KUKA KRL program: ps_b_lta_geo_c03.src, ps_b_lta_geo_c03.dat

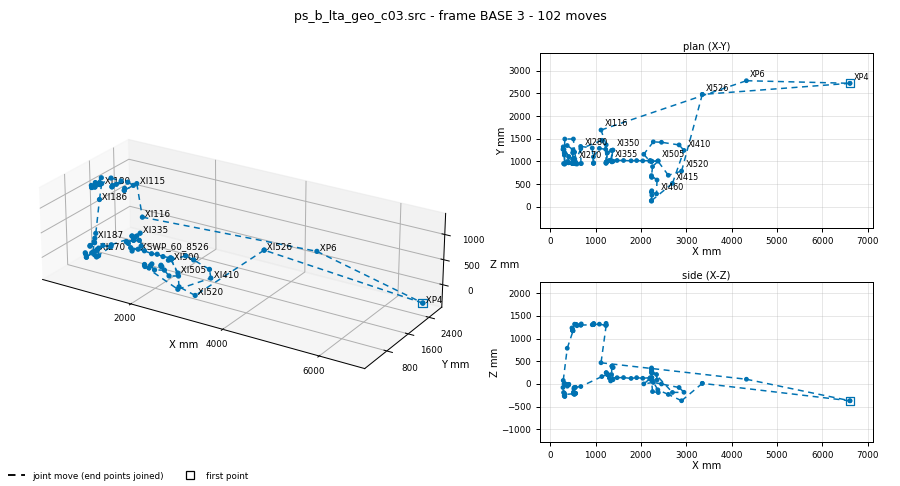
[picture p0: tool path of ps_b_lta_geo_c03.src in frame BASE 3, 102 of 102 moves have a stored position in this frame; points joined in program order, loops and branches not executed]
--- ps_b_lta_geo_c03.src ---
&ACCESS RVO1
&COMMENT Solda Atego LTB
&PARAM DISKPATH = KRC:\R1\Program\OLP
DEF ps_b_lta_geo_c03( )
;FOLD INI
;FOLD SPOTTECH INI
USERSPOT(#INIT)
;ENDFOLD (SPOTTECH INI)
;FOLD GRIPPERTECH INI
USER_GRP(0,DUMMY,DUMMY,GDEFAULT)
;ENDFOLD (GRIPPERTECH INI)
  ;FOLD USER INI
    ;Make your modifications here

  ;ENDFOLD (USER INI)
;ENDFOLD (INI)

; Caracterizacao dos meios de producao
; Changes: Solda Geometria - ATEGO LTB
; Versao Atual:05/01/2016
; Ferramenta: Gun C3
; Name: P13.050-R2
; optimised

chk_w4_wechs_ok( )      ; CHECK GUN C3

;FOLD PTP P4 CONT Vel=100 % PDAT5 Tool[4]:Gun C3 Base[3]:Atego/Axor;%{PE}%R 8.2.20,%MKUKATPBASIS,%CMOVE,%VPTP,%P 1:PTP, 2:P4, 3:C_DIS, 5:100, 7:PDAT5
$BWDSTART=FALSE
PDAT_ACT=PPDAT5
FDAT_ACT=FP4
BAS(#PTP_PARAMS,100)
PTP XP4 C_DIS
;ENDFOLD

if MaxStandMenge (3) then
 MaxStandmengeErreicht (3)
endif

IF (NOT(GHOST())) THEN
if FraesAnf (3) then
 e_fraes4 ()
endif
ENDIF

;FOLD PTP l526 CONT Vel=100 % P_OLP71 Tool[4]:Gun C3 Base[3]:Atego/Axor;%{PE}%R 8.2.20,%MKUKATPBASIS,%CMOVE,%VPTP,%P 1:PTP, 2:l526, 3:C_DIS, 5:100, 7:P_OLP71
$BWDSTART=FALSE
PDAT_ACT=PP_OLP71
FDAT_ACT=Fl526
BAS(#PTP_PARAMS,100)
PTP Xl526 C_DIS
;ENDFOLD

; AGUARDA LIBERACAO PARA SOLDAR GEOMETRIA
;FOLD OUT 3338 'R2 solda geometria Ok' State=FALSE ;%{PE}%R 8.2.20,%MKUKATPBASIS,%COUT,%VOUTX,%P 2:3338, 3:R2 solda geometria Ok, 5:FALSE, 6:
$OUT[3338]=FALSE
;ENDFOLD
;FOLD OUT 3348 'Fora area GEOBOX' State=FALSE ;%{PE}%R 8.2.20,%MKUKATPBASIS,%COUT,%VOUTX,%P 2:3348, 3:Fora area GEOBOX, 5:FALSE, 6:
$OUT[3348]=FALSE
;ENDFOLD
;FOLD OUT 3376 'Lib. p/ soldar Geo Axor/Atego' State=TRUE ;%{PE}%R 8.2.20,%MKUKATPBASIS,%COUT,%VOUTX,%P 2:3376, 3:Lib. p/ soldar Geo Axor/Atego, 5:TRUE, 6:
$OUT[3376]=TRUE
;ENDFOLD
;FOLD WAIT FOR ( IN 3376 'Lib. p/ soldar Geo Axor/Atego' );%{PE}%R 8.2.20,%MKUKATPBASIS,%CEXT_WAIT_FOR,%VEXT_WAIT_FOR,%P 2:, 4:, 5:$IN, 6:3376, 7:Lib. p/ soldar Geo Axor/Atego, 9:
WAIT FOR  ( $IN[3376] )
;ENDFOLD
;FOLD OUT 3376 'Lib. p/ soldar Geo Axor/Atego' State=FALSE ;%{PE}%R 8.2.20,%MKUKATPBASIS,%COUT,%VOUTX,%P 2:3376, 3:Lib. p/ soldar Geo Axor/Atego, 5:FALSE, 6:
$OUT[3376]=FALSE
;ENDFOLD

; LIGA INTERTRAVAMENTO 1 C/ R1
;FOLD Collision.Monitoring_1_On ;%{PE}%MKUKATPUSER
COLLSTOP( 1, 1 ) ;Interrupt-Controlled
;ENDFOLD

; LIGA INTERTRAVAMENTO 4 C/ R4
;FOLD Collision.Monitoring_4_On ;%{PE}%MKUKATPUSER
COLLSTOP( 4, 1 ) ;Interrupt-Controlled
;ENDFOLD

; LIGA INTERTRAVAMENTO 12 C/ R1
;FOLD Collision.Monitoring_AREA_6_On ;%{PE}%MKUKATPUSER
COLLSTOP( 12, 1 ) ;not Interrupt-Controlled
;ENDFOLD

;FOLD PTP l527 CONT Vel=100 % xlarge Tool[4]:Gun C3 Base[3]:Atego/Axor;%{PE}%R 8.2.20,%MKUKATPBASIS,%CMOVE,%VPTP,%P 1:PTP, 2:l527, 3:C_DIS, 5:100, 7:xlarge
$BWDSTART=FALSE
PDAT_ACT=Pxlarge
FDAT_ACT=Fl527
BAS(#PTP_PARAMS,100)
PTP Xl527 C_DIS
;ENDFOLD
;FOLD PTP l520 CONT Vel=100 % xlarge Tool[4]:Gun C3 Base[3]:Atego/Axor;%{PE}%R 8.2.20,%MKUKATPBASIS,%CMOVE,%VPTP,%P 1:PTP, 2:l520, 3:C_DIS, 5:100, 7:xlarge
$BWDSTART=FALSE
PDAT_ACT=Pxlarge
FDAT_ACT=Fl520
BAS(#PTP_PARAMS,100)
PTP Xl520 C_DIS
;ENDFOLD
;FOLD PTP l515 CONT Vel=100 % medium Tool[4]:Gun C3 Base[3]:Atego/Axor;%{PE}%R 8.2.20,%MKUKATPBASIS,%CMOVE,%VPTP,%P 1:PTP, 2:l515, 3:C_DIS, 5:100, 7:medium
$BWDSTART=FALSE
PDAT_ACT=Pmedium
FDAT_ACT=Fl515
BAS(#PTP_PARAMS,100)
PTP Xl515 C_DIS
;ENDFOLD
;FOLD PTP l505 CONT Vel=100 % small Tool[4]:Gun C3 Base[3]:Atego/Axor;%{PE}%R 8.2.20,%MKUKATPBASIS,%CMOVE,%VPTP,%P 1:PTP, 2:l505, 3:C_DIS, 5:100, 7:small
$BWDSTART=FALSE
PDAT_ACT=Psmall
FDAT_ACT=Fl505
BAS(#PTP_PARAMS,100)
PTP Xl505 C_DIS
;ENDFOLD
;FOLD PTP l500 CONT Vel=100 % fin Tool[4]:Gun C3 Base[3]:Atego/Axor;%{PE}%R 8.2.20,%MKUKATPBASIS,%CMOVE,%VPTP,%P 1:PTP, 2:l500, 3:C_DIS, 5:100, 7:fin
$BWDSTART=FALSE
PDAT_ACT=Pfin
FDAT_ACT=Fl500
BAS(#PTP_PARAMS,100)
PTP Xl500 C_DIS
;ENDFOLD

;FOLD ; SWP_60_9492;%{PE}%R 8.2.20,%MKUKATPBASIS,%CCOMMENT,%VNORMAL,%P 2:SWP_60_9492
;ENDFOLD
;FOLD PTP SWP_60_9492 vmax SPOT Gun=3 RETR OPN PgNo1=199 ACTIVE=1 Tool[4]:Gun C3 Base[3]:Atego/Axor;%{PE}%R 8.2.2,%MKUKATPSPOT,%CSPOT,%VPTP,%P 1:PTP, 2:SWP_60_9492, 3:, 5:100, 7:vmax, 10:3, 12:#FIRST, 14:#OPN, 16:199, 18:1, 20:0, 22:0, 24:1, 25:NORMAL
$BWDSTART=FALSE
PDAT_ACT=Pvmax
FDAT_ACT=FSWP_60_9492
BAS(#PTP_PARAMS,Pvmax.VEL)
S_ACT.GUN=3
S_ACT.PAIR=SDEFAULT.PAIR
S_ACT.RETR=#OPN
S_ACT.CLO_TM=1
S_ACT.PGNO1=199
S_ACT.PGNO2=SDEFAULT.PGNO2
S_ACT.PRESS1=SDEFAULT.PRESS1
S_ACT.PRESS2=SDEFAULT.PRESS2
S_READY=FALSE
PTP XSWP_60_9492
USERSPOT(#SPOT, S_ACT)
WAIT FOR S_READY
;ENDFOLD

;FOLD PTP l495 CONT Vel=100 % fin Tool[4]:Gun C3 Base[3]:Atego/Axor;%{PE}%R 8.2.20,%MKUKATPBASIS,%CMOVE,%VPTP,%P 1:PTP, 2:l495, 3:C_DIS, 5:100, 7:fin
$BWDSTART=FALSE
PDAT_ACT=Pfin
FDAT_ACT=Fl495
BAS(#PTP_PARAMS,100)
PTP Xl495 C_DIS
;ENDFOLD
;FOLD PTP l490 CONT Vel=100 % small Tool[4]:Gun C3 Base[3]:Atego/Axor;%{PE}%R 8.2.20,%MKUKATPBASIS,%CMOVE,%VPTP,%P 1:PTP, 2:l490, 3:C_DIS, 5:100, 7:small
$BWDSTART=FALSE
PDAT_ACT=Psmall
FDAT_ACT=Fl490
BAS(#PTP_PARAMS,100)
PTP Xl490 C_DIS
;ENDFOLD
;FOLD PTP l480 CONT Vel=100 % small Tool[4]:Gun C3 Base[3]:Atego/Axor;%{PE}%R 8.2.20,%MKUKATPBASIS,%CMOVE,%VPTP,%P 1:PTP, 2:l480, 3:C_DIS, 5:100, 7:small
$BWDSTART=FALSE
PDAT_ACT=Psmall
FDAT_ACT=Fl480
BAS(#PTP_PARAMS,100)
PTP Xl480 C_DIS
;ENDFOLD
;FOLD PTP l475 CONT Vel=100 % fin Tool[4]:Gun C3 Base[3]:Atego/Axor;%{PE}%R 8.2.20,%MKUKATPBASIS,%CMOVE,%VPTP,%P 1:PTP, 2:l475, 3:C_DIS, 5:100, 7:fin
$BWDSTART=FALSE
PDAT_ACT=Pfin
FDAT_ACT=Fl475
BAS(#PTP_PARAMS,100)
PTP Xl475 C_DIS
;ENDFOLD

;FOLD ; SWP_60_9476;%{PE}%R 8.2.20,%MKUKATPBASIS,%CCOMMENT,%VNORMAL,%P 2:SWP_60_9476
;ENDFOLD
;FOLD PTP SWP_60_9476 vmax SPOT Gun=3 RETR CLS PgNo1=199 ACTIVE=1 Tool[4]:Gun C3 Base[3]:Atego/Axor;%{PE}%R 8.2.2,%MKUKATPSPOT,%CSPOT,%VPTP,%P 1:PTP, 2:SWP_60_9476, 3:, 5:100, 7:vmax, 10:3, 12:#FIRST, 14:#CLO, 16:199, 18:1, 20:0, 22:0, 24:1, 25:NORMAL
$BWDSTART=FALSE
PDAT_ACT=Pvmax
FDAT_ACT=FSWP_60_9476
BAS(#PTP_PARAMS,Pvmax.VEL)
S_ACT.GUN=3
S_ACT.PAIR=SDEFAULT.PAIR
S_ACT.RETR=#CLO
S_ACT.CLO_TM=1
S_ACT.PGNO1=199
S_ACT.PGNO2=SDEFAULT.PGNO2
S_ACT.PRESS1=SDEFAULT.PRESS1
S_ACT.PRESS2=SDEFAULT.PRESS2
S_READY=FALSE
PTP XSWP_60_9476
USERSPOT(#SPOT, S_ACT)
WAIT FOR S_READY
;ENDFOLD

;FOLD PTP l470 CONT Vel=100 % small Tool[4]:Gun C3 Base[3]:Atego/Axor;%{PE}%R 8.2.20,%MKUKATPBASIS,%CMOVE,%VPTP,%P 1:PTP, 2:l470, 3:C_DIS, 5:100, 7:small
$BWDSTART=FALSE
PDAT_ACT=Psmall
FDAT_ACT=Fl470
BAS(#PTP_PARAMS,100)
PTP Xl470 C_DIS
;ENDFOLD
;FOLD PTP l465 CONT Vel=100 % medium Tool[4]:Gun C3 Base[3]:Atego/Axor;%{PE}%R 8.2.20,%MKUKATPBASIS,%CMOVE,%VPTP,%P 1:PTP, 2:l465, 3:C_DIS, 5:100, 7:medium
$BWDSTART=FALSE
PDAT_ACT=Pmedium
FDAT_ACT=Fl465
BAS(#PTP_PARAMS,100)
PTP Xl465 C_DIS
;ENDFOLD
;FOLD PTP l460 CONT Vel=100 % medium Tool[4]:Gun C3 Base[3]:Atego/Axor;%{PE}%R 8.2.20,%MKUKATPBASIS,%CMOVE,%VPTP,%P 1:PTP, 2:l460, 3:C_DIS, 5:100, 7:medium
$BWDSTART=FALSE
PDAT_ACT=Pmedium
FDAT_ACT=Fl460
BAS(#PTP_PARAMS,100)
PTP Xl460 C_DIS
;ENDFOLD
;FOLD PTP l450 CONT Vel=100 % fin Tool[4]:Gun C3 Base[3]:Atego/Axor;%{PE}%R 8.2.20,%MKUKATPBASIS,%CMOVE,%VPTP,%P 1:PTP, 2:l450, 3:C_DIS, 5:100, 7:fin
$BWDSTART=FALSE
PDAT_ACT=Pfin
FDAT_ACT=Fl450
BAS(#PTP_PARAMS,100)
PTP Xl450 C_DIS
;ENDFOLD

;FOLD ; SWP_60_9472;%{PE}%R 8.2.20,%MKUKATPBASIS,%CCOMMENT,%VNORMAL,%P 2:SWP_60_9472
;ENDFOLD
;FOLD PTP SWP_60_9472 vmax SPOT Gun=3 RETR CLS PgNo1=199 ACTIVE=1 Tool[4]:Gun C3 Base[3]:Atego/Axor;%{PE}%R 8.2.2,%MKUKATPSPOT,%CSPOT,%VPTP,%P 1:PTP, 2:SWP_60_9472, 3:, 5:100, 7:vmax, 10:3, 12:#FIRST, 14:#CLO, 16:199, 18:1, 20:0, 22:0, 24:1, 25:NORMAL
$BWDSTART=FALSE
PDAT_ACT=Pvmax
FDAT_ACT=FSWP_60_9472
BAS(#PTP_PARAMS,Pvmax.VEL)
S_ACT.GUN=3
S_ACT.PAIR=SDEFAULT.PAIR
S_ACT.RETR=#CLO
S_ACT.CLO_TM=1
S_ACT.PGNO1=199
S_ACT.PGNO2=SDEFAULT.PGNO2
S_ACT.PRESS1=SDEFAULT.PRESS1
S_ACT.PRESS2=SDEFAULT.PRESS2
S_READY=FALSE
PTP XSWP_60_9472
USERSPOT(#SPOT, S_ACT)
WAIT FOR S_READY
;ENDFOLD


;FOLD PTP l107 CONT Vel=100 % small Tool[4]:Gun C3 Base[3]:Atego/Axor;%{PE}%R 8.2.20,%MKUKATPBASIS,%CMOVE,%VPTP,%P 1:PTP, 2:l107, 3:C_DIS, 5:100, 7:small
$BWDSTART=FALSE
PDAT_ACT=Psmall
FDAT_ACT=Fl107
BAS(#PTP_PARAMS,100)
PTP Xl107 C_DIS
;ENDFOLD
;FOLD PTP l106 CONT Vel=100 % fin Tool[4]:Gun C3 Base[3]:Atego/Axor;%{PE}%R 8.2.20,%MKUKATPBASIS,%CMOVE,%VPTP,%P 1:PTP, 2:l106, 3:C_DIS, 5:100, 7:fin
$BWDSTART=FALSE
PDAT_ACT=Pfin
FDAT_ACT=Fl106
BAS(#PTP_PARAMS,100)
PTP Xl106 C_DIS
;ENDFOLD


;FOLD ; SWP_60_9462;%{PE}%R 8.2.20,%MKUKATPBASIS,%CCOMMENT,%VNORMAL,%P 2:SWP_60_9462
;ENDFOLD
;FOLD PTP SWP_60_9462 vmax SPOT Gun=3 RETR CLS PgNo1=199 ACTIVE=1 Tool[4]:Gun C3 Base[3]:Atego/Axor;%{PE}%R 8.2.2,%MKUKATPSPOT,%CSPOT,%VPTP,%P 1:PTP, 2:SWP_60_9462, 3:, 5:100, 7:vmax, 10:3, 12:#FIRST, 14:#CLO, 16:199, 18:1, 20:0, 22:0, 24:1, 25:NORMAL
$BWDSTART=FALSE
PDAT_ACT=Pvmax
FDAT_ACT=FSWP_60_9462
BAS(#PTP_PARAMS,Pvmax.VEL)
S_ACT.GUN=3
S_ACT.PAIR=SDEFAULT.PAIR
S_ACT.RETR=#CLO
S_ACT.CLO_TM=1
S_ACT.PGNO1=199
S_ACT.PGNO2=SDEFAULT.PGNO2
S_ACT.PRESS1=SDEFAULT.PRESS1
S_ACT.PRESS2=SDEFAULT.PRESS2
S_READY=FALSE
PTP XSWP_60_9462
USERSPOT(#SPOT, S_ACT)
WAIT FOR S_READY
;ENDFOLD

;FOLD PTP l420 CONT Vel=100 % P_OLP48 Tool[4]:Gun C3 Base[3]:Atego/Axor;%{PE}%R 8.2.20,%MKUKATPBASIS,%CMOVE,%VPTP,%P 1:PTP, 2:l420, 3:C_DIS, 5:100, 7:P_OLP48
$BWDSTART=FALSE
PDAT_ACT=PP_OLP48
FDAT_ACT=Fl420
BAS(#PTP_PARAMS,100)
PTP Xl420 C_DIS
;ENDFOLD
;FOLD PTP l415 CONT Vel=100 % xlarge Tool[4]:Gun C3 Base[3]:Atego/Axor;%{PE}%R 8.2.20,%MKUKATPBASIS,%CMOVE,%VPTP,%P 1:PTP, 2:l415, 3:C_DIS, 5:100, 7:xlarge
$BWDSTART=FALSE
PDAT_ACT=Pxlarge
FDAT_ACT=Fl415
BAS(#PTP_PARAMS,100)
PTP Xl415 C_DIS
;ENDFOLD
;FOLD PTP l410 CONT Vel=100 % xlarge Tool[4]:Gun C3 Base[3]:Atego/Axor;%{PE}%R 8.2.20,%MKUKATPBASIS,%CMOVE,%VPTP,%P 1:PTP, 2:l410, 3:C_DIS, 5:100, 7:xlarge
$BWDSTART=FALSE
PDAT_ACT=Pxlarge
FDAT_ACT=Fl410
BAS(#PTP_PARAMS,100)
PTP Xl410 C_DIS
;ENDFOLD
;FOLD PTP l405 CONT Vel=100 % xlarge Tool[4]:Gun C3 Base[3]:Atego/Axor;%{PE}%R 8.2.20,%MKUKATPBASIS,%CMOVE,%VPTP,%P 1:PTP, 2:l405, 3:C_DIS, 5:100, 7:xlarge
$BWDSTART=FALSE
PDAT_ACT=Pxlarge
FDAT_ACT=Fl405
BAS(#PTP_PARAMS,100)
PTP Xl405 C_DIS
;ENDFOLD
;FOLD PTP l400 CONT Vel=100 % medium Tool[4]:Gun C3 Base[3]:Atego/Axor;%{PE}%R 8.2.20,%MKUKATPBASIS,%CMOVE,%VPTP,%P 1:PTP, 2:l400, 3:C_DIS, 5:100, 7:medium
$BWDSTART=FALSE
PDAT_ACT=Pmedium
FDAT_ACT=Fl400
BAS(#PTP_PARAMS,100)
PTP Xl400 C_DIS
;ENDFOLD
;FOLD PTP l395 CONT Vel=100 % xlarge Tool[4]:Gun C3 Base[3]:Atego/Axor;%{PE}%R 8.2.20,%MKUKATPBASIS,%CMOVE,%VPTP,%P 1:PTP, 2:l395, 3:C_DIS, 5:100, 7:xlarge
$BWDSTART=FALSE
PDAT_ACT=Pxlarge
FDAT_ACT=Fl395
BAS(#PTP_PARAMS,100)
PTP Xl395 C_DIS
;ENDFOLD
;FOLD PTP l390 CONT Vel=100 % medium Tool[4]:Gun C3 Base[3]:Atego/Axor;%{PE}%R 8.2.20,%MKUKATPBASIS,%CMOVE,%VPTP,%P 1:PTP, 2:l390, 3:C_DIS, 5:100, 7:medium
$BWDSTART=FALSE
PDAT_ACT=Pmedium
FDAT_ACT=Fl390
BAS(#PTP_PARAMS,100)
PTP Xl390 C_DIS
;ENDFOLD
;FOLD PTP l385 CONT Vel=100 % fin Tool[4]:Gun C3 Base[3]:Atego/Axor;%{PE}%R 8.2.20,%MKUKATPBASIS,%CMOVE,%VPTP,%P 1:PTP, 2:l385, 3:C_DIS, 5:100, 7:fin
$BWDSTART=FALSE
PDAT_ACT=Pfin
FDAT_ACT=Fl385
BAS(#PTP_PARAMS,100)
PTP Xl385 C_DIS
;ENDFOLD

;FOLD ; SWP_60_8494;%{PE}%R 8.2.20,%MKUKATPBASIS,%CCOMMENT,%VNORMAL,%P 2:SWP_60_8494
;ENDFOLD
;FOLD PTP SWP_60_8494 vmax SPOT Gun=3 RETR CLS PgNo1=211 ACTIVE=1 Tool[4]:Gun C3 Base[3]:Atego/Axor;%{PE}%R 8.2.2,%MKUKATPSPOT,%CSPOT,%VPTP,%P 1:PTP, 2:SWP_60_8494, 3:, 5:100, 7:vmax, 10:3, 12:#FIRST, 14:#CLO, 16:211, 18:1, 20:0, 22:0, 24:1, 25:NORMAL
$BWDSTART=FALSE
PDAT_ACT=Pvmax
FDAT_ACT=FSWP_60_8494
BAS(#PTP_PARAMS,Pvmax.VEL)
S_ACT.GUN=3
S_ACT.PAIR=SDEFAULT.PAIR
S_ACT.RETR=#CLO
S_ACT.CLO_TM=1
S_ACT.PGNO1=211
S_ACT.PGNO2=SDEFAULT.PGNO2
S_ACT.PRESS1=SDEFAULT.PRESS1
S_ACT.PRESS2=SDEFAULT.PRESS2
S_READY=FALSE
PTP XSWP_60_8494
USERSPOT(#SPOT, S_ACT)
WAIT FOR S_READY
;ENDFOLD

; DESLIGA INTERTRAVAMENTO 12 C/ R1
;FOLD Collision.Monitoring_AREA_6_Off . ;%{PE}%MKUKATPUSER
COLLSTOP( 12, 2+0 )
;ENDFOLD

;FOLD PTP P5 CONT Vel=100 % large Tool[4]:Gun C3 Base[3]:Atego/Axor;%{PE}%R 8.2.20,%MKUKATPBASIS,%CMOVE,%VPTP,%P 1:PTP, 2:P5, 3:C_DIS, 5:100, 7:large
$BWDSTART=FALSE
PDAT_ACT=Plarge
FDAT_ACT=FP5
BAS(#PTP_PARAMS,100)
PTP XP5 C_DIS
;ENDFOLD

;FOLD ; SWP_60_8506;%{PE}%R 8.2.20,%MKUKATPBASIS,%CCOMMENT,%VNORMAL,%P 2:SWP_60_8506
;ENDFOLD
;FOLD PTP SWP_60_8506 vmax SPOT Gun=3 RETR CLS PgNo1=203 ACTIVE=1 Tool[4]:Gun C3 Base[3]:Atego/Axor;%{PE}%R 8.2.2,%MKUKATPSPOT,%CSPOT,%VPTP,%P 1:PTP, 2:SWP_60_8506, 3:, 5:100, 7:vmax, 10:3, 12:#FIRST, 14:#CLO, 16:203, 18:1, 20:0, 22:0, 24:1, 25:NORMAL
$BWDSTART=FALSE
PDAT_ACT=Pvmax
FDAT_ACT=FSWP_60_8506
BAS(#PTP_PARAMS,Pvmax.VEL)
S_ACT.GUN=3
S_ACT.PAIR=SDEFAULT.PAIR
S_ACT.RETR=#CLO
S_ACT.CLO_TM=1
S_ACT.PGNO1=203
S_ACT.PGNO2=SDEFAULT.PGNO2
S_ACT.PRESS1=SDEFAULT.PRESS1
S_ACT.PRESS2=SDEFAULT.PRESS2
S_READY=FALSE
PTP XSWP_60_8506
USERSPOT(#SPOT, S_ACT)
WAIT FOR S_READY
;ENDFOLD

;FOLD PTP l380 CONT Vel=100 % large Tool[4]:Gun C3 Base[3]:Atego/Axor;%{PE}%R 8.2.20,%MKUKATPBASIS,%CMOVE,%VPTP,%P 1:PTP, 2:l380, 3:C_DIS, 5:100, 7:large
$BWDSTART=FALSE
PDAT_ACT=Plarge
FDAT_ACT=Fl380
BAS(#PTP_PARAMS,100)
PTP Xl380 C_DIS
;ENDFOLD

;FOLD ; SWP_60_8518;%{PE}%R 8.2.20,%MKUKATPBASIS,%CCOMMENT,%VNORMAL,%P 2:SWP_60_8518
;ENDFOLD
;FOLD PTP SWP_60_8518 vmax SPOT Gun=3 RETR CLS PgNo1=212 ACTIVE=1 Tool[4]:Gun C3 Base[3]:Atego/Axor;%{PE}%R 8.2.2,%MKUKATPSPOT,%CSPOT,%VPTP,%P 1:PTP, 2:SWP_60_8518, 3:, 5:100, 7:vmax, 10:3, 12:#FIRST, 14:#CLO, 16:212, 18:1, 20:0, 22:0, 24:1, 25:NORMAL
$BWDSTART=FALSE
PDAT_ACT=Pvmax
FDAT_ACT=FSWP_60_8518
BAS(#PTP_PARAMS,Pvmax.VEL)
S_ACT.GUN=3
S_ACT.PAIR=SDEFAULT.PAIR
S_ACT.RETR=#CLO
S_ACT.CLO_TM=1
S_ACT.PGNO1=212
S_ACT.PGNO2=SDEFAULT.PGNO2
S_ACT.PRESS1=SDEFAULT.PRESS1
S_ACT.PRESS2=SDEFAULT.PRESS2
S_READY=FALSE
PTP XSWP_60_8518
USERSPOT(#SPOT, S_ACT)
WAIT FOR S_READY
;ENDFOLD

;FOLD ; SWP_60_8526;%{PE}%R 8.2.20,%MKUKATPBASIS,%CCOMMENT,%VNORMAL,%P 2:SWP_60_8526
;ENDFOLD
;FOLD PTP SWP_60_8526 vmax SPOT Gun=3 RETR CLS PgNo1=206 ACTIVE=1 Tool[4]:Gun C3 Base[3]:Atego/Axor;%{PE}%R 8.2.2,%MKUKATPSPOT,%CSPOT,%VPTP,%P 1:PTP, 2:SWP_60_8526, 3:, 5:100, 7:vmax, 10:3, 12:#FIRST, 14:#CLO, 16:206, 18:1, 20:0, 22:0, 24:1, 25:NORMAL
$BWDSTART=FALSE
PDAT_ACT=Pvmax
FDAT_ACT=FSWP_60_8526
BAS(#PTP_PARAMS,Pvmax.VEL)
S_ACT.GUN=3
S_ACT.PAIR=SDEFAULT.PAIR
S_ACT.RETR=#CLO
S_ACT.CLO_TM=1
S_ACT.PGNO1=206
S_ACT.PGNO2=SDEFAULT.PGNO2
S_ACT.PRESS1=SDEFAULT.PRESS1
S_ACT.PRESS2=SDEFAULT.PRESS2
S_READY=FALSE
PTP XSWP_60_8526
USERSPOT(#SPOT, S_ACT)
WAIT FOR S_READY
;ENDFOLD

;FOLD ; SWP_60_8534;%{PE}%R 8.2.20,%MKUKATPBASIS,%CCOMMENT,%VNORMAL,%P 2:SWP_60_8534
;ENDFOLD
;FOLD PTP SWP_60_8534 vmax SPOT Gun=3 RETR CLS PgNo1=206 ACTIVE=1 Tool[4]:Gun C3 Base[3]:Atego/Axor;%{PE}%R 8.2.2,%MKUKATPSPOT,%CSPOT,%VPTP,%P 1:PTP, 2:SWP_60_8534, 3:, 5:100, 7:vmax, 10:3, 12:#FIRST, 14:#CLO, 16:206, 18:1, 20:0, 22:0, 24:1, 25:NORMAL
$BWDSTART=FALSE
PDAT_ACT=Pvmax
FDAT_ACT=FSWP_60_8534
BAS(#PTP_PARAMS,Pvmax.VEL)
S_ACT.GUN=3
S_ACT.PAIR=SDEFAULT.PAIR
S_ACT.RETR=#CLO
S_ACT.CLO_TM=1
S_ACT.PGNO1=206
S_ACT.PGNO2=SDEFAULT.PGNO2
S_ACT.PRESS1=SDEFAULT.PRESS1
S_ACT.PRESS2=SDEFAULT.PRESS2
S_READY=FALSE
PTP XSWP_60_8534
USERSPOT(#SPOT, S_ACT)
WAIT FOR S_READY
;ENDFOLD

;FOLD PTP l355 CONT Vel=100 % small Tool[4]:Gun C3 Base[3]:Atego/Axor;%{PE}%R 8.2.20,%MKUKATPBASIS,%CMOVE,%VPTP,%P 1:PTP, 2:l355, 3:C_DIS, 5:100, 7:small
$BWDSTART=FALSE
PDAT_ACT=Psmall
FDAT_ACT=Fl355
BAS(#PTP_PARAMS,100)
PTP Xl355 C_DIS
;ENDFOLD
;FOLD PTP l350 CONT Vel=100 % large Tool[4]:Gun C3 Base[3]:Atego/Axor;%{PE}%R 8.2.20,%MKUKATPBASIS,%CMOVE,%VPTP,%P 1:PTP, 2:l350, 3:C_DIS, 5:100, 7:large
$BWDSTART=FALSE
PDAT_ACT=Plarge
FDAT_ACT=Fl350
BAS(#PTP_PARAMS,100)
PTP Xl350 C_DIS
;ENDFOLD
;FOLD PTP l335 CONT Vel=100 % medium Tool[4]:Gun C3 Base[3]:Atego/Axor;%{PE}%R 8.2.20,%MKUKATPBASIS,%CMOVE,%VPTP,%P 1:PTP, 2:l335, 3:C_DIS, 5:100, 7:medium
$BWDSTART=FALSE
PDAT_ACT=Pmedium
FDAT_ACT=Fl335
BAS(#PTP_PARAMS,100)
PTP Xl335 C_DIS
;ENDFOLD
;FOLD PTP l330 CONT Vel=100 % fin Tool[4]:Gun C3 Base[3]:Atego/Axor;%{PE}%R 8.2.20,%MKUKATPBASIS,%CMOVE,%VPTP,%P 1:PTP, 2:l330, 3:C_DIS, 5:100, 7:fin
$BWDSTART=FALSE
PDAT_ACT=Pfin
FDAT_ACT=Fl330
BAS(#PTP_PARAMS,100)
PTP Xl330 C_DIS
;ENDFOLD

;FOLD ; SWP_60_8554;%{PE}%R 8.2.20,%MKUKATPBASIS,%CCOMMENT,%VNORMAL,%P 2:SWP_60_8554
;ENDFOLD
;FOLD PTP SWP_60_8554 vmax SPOT Gun=3 RETR CLS PgNo1=197 ACTIVE=1 Tool[4]:Gun C3 Base[3]:Atego/Axor;%{PE}%R 8.2.2,%MKUKATPSPOT,%CSPOT,%VPTP,%P 1:PTP, 2:SWP_60_8554, 3:, 5:100, 7:vmax, 10:3, 12:#FIRST, 14:#CLO, 16:197, 18:1, 20:0, 22:0, 24:1, 25:NORMAL
$BWDSTART=FALSE
PDAT_ACT=Pvmax
FDAT_ACT=FSWP_60_8554
BAS(#PTP_PARAMS,Pvmax.VEL)
S_ACT.GUN=3
S_ACT.PAIR=SDEFAULT.PAIR
S_ACT.RETR=#CLO
S_ACT.CLO_TM=1
S_ACT.PGNO1=197
S_ACT.PGNO2=SDEFAULT.PGNO2
S_ACT.PRESS1=SDEFAULT.PRESS1
S_ACT.PRESS2=SDEFAULT.PRESS2
S_READY=FALSE
PTP XSWP_60_8554
USERSPOT(#SPOT, S_ACT)
WAIT FOR S_READY
;ENDFOLD

;FOLD PTP l325 CONT Vel=100 % fin Tool[4]:Gun C3 Base[3]:Atego/Axor;%{PE}%R 8.2.20,%MKUKATPBASIS,%CMOVE,%VPTP,%P 1:PTP, 2:l325, 3:C_DIS, 5:100, 7:fin
$BWDSTART=FALSE
PDAT_ACT=Pfin
FDAT_ACT=Fl325
BAS(#PTP_PARAMS,100)
PTP Xl325 C_DIS
;ENDFOLD
;FOLD PTP l320 CONT Vel=100 % small Tool[4]:Gun C3 Base[3]:Atego/Axor;%{PE}%R 8.2.20,%MKUKATPBASIS,%CMOVE,%VPTP,%P 1:PTP, 2:l320, 3:C_DIS, 5:100, 7:small
$BWDSTART=FALSE
PDAT_ACT=Psmall
FDAT_ACT=Fl320
BAS(#PTP_PARAMS,100)
PTP Xl320 C_DIS
;ENDFOLD
;FOLD PTP l310 CONT Vel=100 % small Tool[4]:Gun C3 Base[3]:Atego/Axor;%{PE}%R 8.2.20,%MKUKATPBASIS,%CMOVE,%VPTP,%P 1:PTP, 2:l310, 3:C_DIS, 5:100, 7:small
$BWDSTART=FALSE
PDAT_ACT=Psmall
FDAT_ACT=Fl310
BAS(#PTP_PARAMS,100)
PTP Xl310 C_DIS
;ENDFOLD
;FOLD PTP l300 CONT Vel=100 % fin Tool[4]:Gun C3 Base[3]:Atego/Axor;%{PE}%R 8.2.20,%MKUKATPBASIS,%CMOVE,%VPTP,%P 1:PTP, 2:l300, 3:C_DIS, 5:100, 7:fin
$BWDSTART=FALSE
PDAT_ACT=Pfin
FDAT_ACT=Fl300
BAS(#PTP_PARAMS,100)
PTP Xl300 C_DIS
;ENDFOLD

;FOLD ; SWP_60_8542;%{PE}%R 8.2.20,%MKUKATPBASIS,%CCOMMENT,%VNORMAL,%P 2:SWP_60_8542
;ENDFOLD
;FOLD PTP SWP_60_8542 vmax SPOT Gun=3 RETR CLS PgNo1=215 ACTIVE=1 Tool[4]:Gun C3 Base[3]:Atego/Axor;%{PE}%R 8.2.2,%MKUKATPSPOT,%CSPOT,%VPTP,%P 1:PTP, 2:SWP_60_8542, 3:, 5:100, 7:vmax, 10:3, 12:#FIRST, 14:#CLO, 16:215, 18:1, 20:0, 22:0, 24:1, 25:NORMAL
$BWDSTART=FALSE
PDAT_ACT=Pvmax
FDAT_ACT=FSWP_60_8542
BAS(#PTP_PARAMS,Pvmax.VEL)
S_ACT.GUN=3
S_ACT.PAIR=SDEFAULT.PAIR
S_ACT.RETR=#CLO
S_ACT.CLO_TM=1
S_ACT.PGNO1=215
S_ACT.PGNO2=SDEFAULT.PGNO2
S_ACT.PRESS1=SDEFAULT.PRESS1
S_ACT.PRESS2=SDEFAULT.PRESS2
S_READY=FALSE
PTP XSWP_60_8542
USERSPOT(#SPOT, S_ACT)
WAIT FOR S_READY
;ENDFOLD

;FOLD PTP l295 CONT Vel=100 % fin Tool[4]:Gun C3 Base[3]:Atego/Axor;%{PE}%R 8.2.20,%MKUKATPBASIS,%CMOVE,%VPTP,%P 1:PTP, 2:l295, 3:C_DIS, 5:100, 7:fin
$BWDSTART=FALSE
PDAT_ACT=Pfin
FDAT_ACT=Fl295
BAS(#PTP_PARAMS,100)
PTP Xl295 C_DIS
;ENDFOLD
;FOLD PTP l290 CONT Vel=100 % small Tool[4]:Gun C3 Base[3]:Atego/Axor;%{PE}%R 8.2.20,%MKUKATPBASIS,%CMOVE,%VPTP,%P 1:PTP, 2:l290, 3:C_DIS, 5:100, 7:small
$BWDSTART=FALSE
PDAT_ACT=Psmall
FDAT_ACT=Fl290
BAS(#PTP_PARAMS,100)
PTP Xl290 C_DIS
;ENDFOLD
;FOLD PTP l285 CONT Vel=100 % large Tool[4]:Gun C3 Base[3]:Atego/Axor;%{PE}%R 8.2.20,%MKUKATPBASIS,%CMOVE,%VPTP,%P 1:PTP, 2:l285, 3:C_DIS, 5:100, 7:large
$BWDSTART=FALSE
PDAT_ACT=Plarge
FDAT_ACT=Fl285
BAS(#PTP_PARAMS,100)
PTP Xl285 C_DIS
;ENDFOLD
;FOLD PTP l280 CONT Vel=100 % medium Tool[4]:Gun C3 Base[3]:Atego/Axor;%{PE}%R 8.2.20,%MKUKATPBASIS,%CMOVE,%VPTP,%P 1:PTP, 2:l280, 3:C_DIS, 5:100, 7:medium
$BWDSTART=FALSE
PDAT_ACT=Pmedium
FDAT_ACT=Fl280
BAS(#PTP_PARAMS,100)
PTP Xl280 C_DIS
;ENDFOLD
;FOLD PTP l270 CONT Vel=100 % fin Tool[4]:Gun C3 Base[3]:Atego/Axor;%{PE}%R 8.2.20,%MKUKATPBASIS,%CMOVE,%VPTP,%P 1:PTP, 2:l270, 3:C_DIS, 5:100, 7:fin
$BWDSTART=FALSE
PDAT_ACT=Pfin
FDAT_ACT=Fl270
BAS(#PTP_PARAMS,100)
PTP Xl270 C_DIS
;ENDFOLD

;FOLD ; SWP_60_8068;%{PE}%R 8.2.20,%MKUKATPBASIS,%CCOMMENT,%VNORMAL,%P 2:SWP_60_8068
;ENDFOLD
;FOLD PTP SWP_60_8068 fin SPOT Gun=3 RETR CLS PgNo1=207 ACTIVE=1 Tool[4]:Gun C3 Base[3]:Atego/Axor;%{PE}%R 8.2.2,%MKUKATPSPOT,%CSPOT,%VPTP,%P 1:PTP, 2:SWP_60_8068, 3:, 5:100, 7:fin, 10:3, 12:#FIRST, 14:#CLO, 16:207, 18:1, 20:0, 22:0, 24:1, 25:NORMAL
$BWDSTART=FALSE
PDAT_ACT=Pfin
FDAT_ACT=FSWP_60_8068
BAS(#PTP_PARAMS,Pfin.VEL)
S_ACT.GUN=3
S_ACT.PAIR=SDEFAULT.PAIR
S_ACT.RETR=#CLO
S_ACT.CLO_TM=1
S_ACT.PGNO1=207
S_ACT.PGNO2=SDEFAULT.PGNO2
S_ACT.PRESS1=SDEFAULT.PRESS1
S_ACT.PRESS2=SDEFAULT.PRESS2
S_READY=FALSE
PTP XSWP_60_8068
USERSPOT(#SPOT, S_ACT)
WAIT FOR S_READY
;ENDFOLD

;FOLD PTP l265 CONT Vel=100 % fin Tool[4]:Gun C3 Base[3]:Atego/Axor;%{PE}%R 8.2.20,%MKUKATPBASIS,%CMOVE,%VPTP,%P 1:PTP, 2:l265, 3:C_DIS, 5:100, 7:fin
$BWDSTART=FALSE
PDAT_ACT=Pfin
FDAT_ACT=Fl265
BAS(#PTP_PARAMS,100)
PTP Xl265 C_DIS
;ENDFOLD
;FOLD PTP l255 CONT Vel=100 % small Tool[4]:Gun C3 Base[3]:Atego/Axor;%{PE}%R 8.2.20,%MKUKATPBASIS,%CMOVE,%VPTP,%P 1:PTP, 2:l255, 3:C_DIS, 5:100, 7:small
$BWDSTART=FALSE
PDAT_ACT=Psmall
FDAT_ACT=Fl255
BAS(#PTP_PARAMS,100)
PTP Xl255 C_DIS
;ENDFOLD
;FOLD PTP l250 CONT Vel=100 % small Tool[4]:Gun C3 Base[3]:Atego/Axor;%{PE}%R 8.2.20,%MKUKATPBASIS,%CMOVE,%VPTP,%P 1:PTP, 2:l250, 3:C_DIS, 5:100, 7:small
$BWDSTART=FALSE
PDAT_ACT=Psmall
FDAT_ACT=Fl250
BAS(#PTP_PARAMS,100)
PTP Xl250 C_DIS
;ENDFOLD
;FOLD PTP l240 CONT Vel=100 % fin Tool[4]:Gun C3 Base[3]:Atego/Axor;%{PE}%R 8.2.20,%MKUKATPBASIS,%CMOVE,%VPTP,%P 1:PTP, 2:l240, 3:C_DIS, 5:100, 7:fin
$BWDSTART=FALSE
PDAT_ACT=Pfin
FDAT_ACT=Fl240
BAS(#PTP_PARAMS,100)
PTP Xl240 C_DIS
;ENDFOLD

;FOLD ; SWP_60_8060;%{PE}%R 8.2.20,%MKUKATPBASIS,%CCOMMENT,%VNORMAL,%P 2:SWP_60_8060
;ENDFOLD
;FOLD PTP SWP_60_8060 vmax SPOT Gun=3 RETR OPN PgNo1=210 ACTIVE=1 Tool[4]:Gun C3 Base[3]:Atego/Axor;%{PE}%R 8.2.2,%MKUKATPSPOT,%CSPOT,%VPTP,%P 1:PTP, 2:SWP_60_8060, 3:, 5:100, 7:vmax, 10:3, 12:#FIRST, 14:#OPN, 16:210, 18:1, 20:0, 22:0, 24:1, 25:NORMAL
$BWDSTART=FALSE
PDAT_ACT=Pvmax
FDAT_ACT=FSWP_60_8060
BAS(#PTP_PARAMS,Pvmax.VEL)
S_ACT.GUN=3
S_ACT.PAIR=SDEFAULT.PAIR
S_ACT.RETR=#OPN
S_ACT.CLO_TM=1
S_ACT.PGNO1=210
S_ACT.PGNO2=SDEFAULT.PGNO2
S_ACT.PRESS1=SDEFAULT.PRESS1
S_ACT.PRESS2=SDEFAULT.PRESS2
S_READY=FALSE
PTP XSWP_60_8060
USERSPOT(#SPOT, S_ACT)
WAIT FOR S_READY
;ENDFOLD

;FOLD PTP l230 CONT Vel=100 % fin Tool[4]:Gun C3 Base[3]:Atego/Axor;%{PE}%R 8.2.20,%MKUKATPBASIS,%CMOVE,%VPTP,%P 1:PTP, 2:l230, 3:C_DIS, 5:100, 7:fin
$BWDSTART=FALSE
PDAT_ACT=Pfin
FDAT_ACT=Fl230
BAS(#PTP_PARAMS,100)
PTP Xl230 C_DIS
;ENDFOLD
;FOLD PTP l225 CONT Vel=100 % medium Tool[4]:Gun C3 Base[3]:Atego/Axor;%{PE}%R 8.2.20,%MKUKATPBASIS,%CMOVE,%VPTP,%P 1:PTP, 2:l225, 3:C_DIS, 5:100, 7:medium
$BWDSTART=FALSE
PDAT_ACT=Pmedium
FDAT_ACT=Fl225
BAS(#PTP_PARAMS,100)
PTP Xl225 C_DIS
;ENDFOLD
;FOLD PTP l220 CONT Vel=100 % medium Tool[4]:Gun C3 Base[3]:Atego/Axor;%{PE}%R 8.2.20,%MKUKATPBASIS,%CMOVE,%VPTP,%P 1:PTP, 2:l220, 3:C_DIS, 5:100, 7:medium
$BWDSTART=FALSE
PDAT_ACT=Pmedium
FDAT_ACT=Fl220
BAS(#PTP_PARAMS,100)
PTP Xl220 C_DIS
;ENDFOLD
;FOLD PTP l215 CONT Vel=100 % small Tool[4]:Gun C3 Base[3]:Atego/Axor;%{PE}%R 8.2.20,%MKUKATPBASIS,%CMOVE,%VPTP,%P 1:PTP, 2:l215, 3:C_DIS, 5:100, 7:small
$BWDSTART=FALSE
PDAT_ACT=Psmall
FDAT_ACT=Fl215
BAS(#PTP_PARAMS,100)
PTP Xl215 C_DIS
;ENDFOLD
;FOLD PTP l210 CONT Vel=100 % small Tool[4]:Gun C3 Base[3]:Atego/Axor;%{PE}%R 8.2.20,%MKUKATPBASIS,%CMOVE,%VPTP,%P 1:PTP, 2:l210, 3:C_DIS, 5:100, 7:small
$BWDSTART=FALSE
PDAT_ACT=Psmall
FDAT_ACT=Fl210
BAS(#PTP_PARAMS,100)
PTP Xl210 C_DIS
;ENDFOLD
;FOLD PTP l205 CONT Vel=100 % fin Tool[4]:Gun C3 Base[3]:Atego/Axor;%{PE}%R 8.2.20,%MKUKATPBASIS,%CMOVE,%VPTP,%P 1:PTP, 2:l205, 3:C_DIS, 5:100, 7:fin
$BWDSTART=FALSE
PDAT_ACT=Pfin
FDAT_ACT=Fl205
BAS(#PTP_PARAMS,100)
PTP Xl205 C_DIS
;ENDFOLD

;FOLD ; SWP_60_8046;%{PE}%R 8.2.20,%MKUKATPBASIS,%CCOMMENT,%VNORMAL,%P 2:SWP_60_8046
;ENDFOLD
;FOLD PTP SWP_60_8046 fin SPOT Gun=3 RETR OPN PgNo1=202 ACTIVE=1 Tool[4]:Gun C3 Base[3]:Atego/Axor;%{PE}%R 8.2.2,%MKUKATPSPOT,%CSPOT,%VPTP,%P 1:PTP, 2:SWP_60_8046, 3:, 5:100, 7:fin, 10:3, 12:#FIRST, 14:#OPN, 16:202, 18:1, 20:0, 22:0, 24:1, 25:NORMAL
$BWDSTART=FALSE
PDAT_ACT=Pfin
FDAT_ACT=FSWP_60_8046
BAS(#PTP_PARAMS,Pfin.VEL)
S_ACT.GUN=3
S_ACT.PAIR=SDEFAULT.PAIR
S_ACT.RETR=#OPN
S_ACT.CLO_TM=1
S_ACT.PGNO1=202
S_ACT.PGNO2=SDEFAULT.PGNO2
S_ACT.PRESS1=SDEFAULT.PRESS1
S_ACT.PRESS2=SDEFAULT.PRESS2
S_READY=FALSE
PTP XSWP_60_8046
USERSPOT(#SPOT, S_ACT)
WAIT FOR S_READY
;ENDFOLD

;FOLD PTP l200 CONT Vel=100 % fin Tool[4]:Gun C3 Base[3]:Atego/Axor;%{PE}%R 8.2.20,%MKUKATPBASIS,%CMOVE,%VPTP,%P 1:PTP, 2:l200, 3:C_DIS, 5:100, 7:fin
$BWDSTART=FALSE
PDAT_ACT=Pfin
FDAT_ACT=Fl200
BAS(#PTP_PARAMS,100)
PTP Xl200 C_DIS
;ENDFOLD
;FOLD PTP l195 CONT Vel=100 % medium Tool[4]:Gun C3 Base[3]:Atego/Axor;%{PE}%R 8.2.20,%MKUKATPBASIS,%CMOVE,%VPTP,%P 1:PTP, 2:l195, 3:C_DIS, 5:100, 7:medium
$BWDSTART=FALSE
PDAT_ACT=Pmedium
FDAT_ACT=Fl195
BAS(#PTP_PARAMS,100)
PTP Xl195 C_DIS
;ENDFOLD
;FOLD PTP l185 CONT Vel=100 % medium Tool[4]:Gun C3 Base[3]:Atego/Axor;%{PE}%R 8.2.20,%MKUKATPBASIS,%CMOVE,%VPTP,%P 1:PTP, 2:l185, 3:C_DIS, 5:100, 7:medium
$BWDSTART=FALSE
PDAT_ACT=Pmedium
FDAT_ACT=Fl185
BAS(#PTP_PARAMS,100)
PTP Xl185 C_DIS
;ENDFOLD
;FOLD PTP l187 CONT Vel=100 % medium Tool[4]:Gun C3 Base[3]:Atego/Axor;%{PE}%R 8.2.20,%MKUKATPBASIS,%CMOVE,%VPTP,%P 1:PTP, 2:l187, 3:C_DIS, 5:100, 7:medium
$BWDSTART=FALSE
PDAT_ACT=Pmedium
FDAT_ACT=Fl187
BAS(#PTP_PARAMS,100)
PTP Xl187 C_DIS
;ENDFOLD
;FOLD PTP l036 CONT Vel=100 % medium Tool[4]:Gun C3 Base[3]:Atego/Axor;%{PE}%R 8.2.20,%MKUKATPBASIS,%CMOVE,%VPTP,%P 1:PTP, 2:l036, 3:C_DIS, 5:100, 7:medium
$BWDSTART=FALSE
PDAT_ACT=Pmedium
FDAT_ACT=Fl036
BAS(#PTP_PARAMS,100)
PTP Xl036 C_DIS
;ENDFOLD
;FOLD PTP l031 CONT Vel=100 % fin Tool[4]:Gun C3 Base[3]:Atego/Axor;%{PE}%R 8.2.20,%MKUKATPBASIS,%CMOVE,%VPTP,%P 1:PTP, 2:l031, 3:C_DIS, 5:100, 7:fin
$BWDSTART=FALSE
PDAT_ACT=Pfin
FDAT_ACT=Fl031
BAS(#PTP_PARAMS,100)
PTP Xl031 C_DIS
;ENDFOLD

;FOLD ; SWP_60_9078;%{PE}%R 8.2.20,%MKUKATPBASIS,%CCOMMENT,%VNORMAL,%P 2:SWP_60_9078
;ENDFOLD
;FOLD PTP SWP_60_9078 vmax SPOT Gun=3 RETR CLS PgNo1=213 ACTIVE=1 Tool[4]:Gun C3 Base[3]:Atego/Axor;%{PE}%R 8.2.2,%MKUKATPSPOT,%CSPOT,%VPTP,%P 1:PTP, 2:SWP_60_9078, 3:, 5:100, 7:vmax, 10:3, 12:#FIRST, 14:#CLO, 16:213, 18:1, 20:0, 22:0, 24:1, 25:NORMAL
$BWDSTART=FALSE
PDAT_ACT=Pvmax
FDAT_ACT=FSWP_60_9078
BAS(#PTP_PARAMS,Pvmax.VEL)
S_ACT.GUN=3
S_ACT.PAIR=SDEFAULT.PAIR
S_ACT.RETR=#CLO
S_ACT.CLO_TM=1
S_ACT.PGNO1=213
S_ACT.PGNO2=SDEFAULT.PGNO2
S_ACT.PRESS1=SDEFAULT.PRESS1
S_ACT.PRESS2=SDEFAULT.PRESS2
S_READY=FALSE
PTP XSWP_60_9078
USERSPOT(#SPOT, S_ACT)
WAIT FOR S_READY
;ENDFOLD

;FOLD PTP l026 CONT Vel=100 % fin Tool[4]:Gun C3 Base[3]:Atego/Axor;%{PE}%R 8.2.20,%MKUKATPBASIS,%CMOVE,%VPTP,%P 1:PTP, 2:l026, 3:C_DIS, 5:100, 7:fin
$BWDSTART=FALSE
PDAT_ACT=Pfin
FDAT_ACT=Fl026
BAS(#PTP_PARAMS,100)
PTP Xl026 C_DIS
;ENDFOLD
;FOLD PTP l021 CONT Vel=100 % medium Tool[4]:Gun C3 Base[3]:Atego/Axor;%{PE}%R 8.2.20,%MKUKATPBASIS,%CMOVE,%VPTP,%P 1:PTP, 2:l021, 3:C_DIS, 5:100, 7:medium
$BWDSTART=FALSE
PDAT_ACT=Pmedium
FDAT_ACT=Fl021
BAS(#PTP_PARAMS,100)
PTP Xl021 C_DIS
;ENDFOLD
;FOLD PTP l188 CONT Vel=100 % medium Tool[4]:Gun C3 Base[3]:Atego/Axor;%{PE}%R 8.2.20,%MKUKATPBASIS,%CMOVE,%VPTP,%P 1:PTP, 2:l188, 3:C_DIS, 5:100, 7:medium
$BWDSTART=FALSE
PDAT_ACT=Pmedium
FDAT_ACT=Fl188
BAS(#PTP_PARAMS,100)
PTP Xl188 C_DIS
;ENDFOLD
;FOLD PTP l186 CONT Vel=100 % large Tool[4]:Gun C3 Base[3]:Atego/Axor;%{PE}%R 8.2.20,%MKUKATPBASIS,%CMOVE,%VPTP,%P 1:PTP, 2:l186, 3:C_DIS, 5:100, 7:large
$BWDSTART=FALSE
PDAT_ACT=Plarge
FDAT_ACT=Fl186
BAS(#PTP_PARAMS,100)
PTP Xl186 C_DIS
;ENDFOLD
;FOLD PTP l180 CONT Vel=100 % medium Tool[4]:Gun C3 Base[3]:Atego/Axor;%{PE}%R 8.2.20,%MKUKATPBASIS,%CMOVE,%VPTP,%P 1:PTP, 2:l180, 3:C_DIS, 5:100, 7:medium
$BWDSTART=FALSE
PDAT_ACT=Pmedium
FDAT_ACT=Fl180
BAS(#PTP_PARAMS,100)
PTP Xl180 C_DIS
;ENDFOLD
;FOLD PTP l175 CONT Vel=100 % small Tool[4]:Gun C3 Base[3]:Atego/Axor;%{PE}%R 8.2.20,%MKUKATPBASIS,%CMOVE,%VPTP,%P 1:PTP, 2:l175, 3:C_DIS, 5:100, 7:small
$BWDSTART=FALSE
PDAT_ACT=Psmall
FDAT_ACT=Fl175
BAS(#PTP_PARAMS,100)
PTP Xl175 C_DIS
;ENDFOLD
;FOLD PTP l170 CONT Vel=100 % fin Tool[4]:Gun C3 Base[3]:Atego/Axor;%{PE}%R 8.2.20,%MKUKATPBASIS,%CMOVE,%VPTP,%P 1:PTP, 2:l170, 3:C_DIS, 5:100, 7:fin
$BWDSTART=FALSE
PDAT_ACT=Pfin
FDAT_ACT=Fl170
BAS(#PTP_PARAMS,100)
PTP Xl170 C_DIS
;ENDFOLD

;FOLD ; SWP_60_8576;%{PE}%R 8.2.20,%MKUKATPBASIS,%CCOMMENT,%VNORMAL,%P 2:SWP_60_8576
;ENDFOLD
;FOLD PTP SWP_60_8576 vmax SPOT Gun=3 RETR CLS PgNo1=209 ACTIVE=1 Tool[4]:Gun C3 Base[3]:Atego/Axor;%{PE}%R 8.2.2,%MKUKATPSPOT,%CSPOT,%VPTP,%P 1:PTP, 2:SWP_60_8576, 3:, 5:100, 7:vmax, 10:3, 12:#FIRST, 14:#CLO, 16:209, 18:1, 20:0, 22:0, 24:1, 25:NORMAL
$BWDSTART=FALSE
PDAT_ACT=Pvmax
FDAT_ACT=FSWP_60_8576
BAS(#PTP_PARAMS,Pvmax.VEL)
S_ACT.GUN=3
S_ACT.PAIR=SDEFAULT.PAIR
S_ACT.RETR=#CLO
S_ACT.CLO_TM=1
S_ACT.PGNO1=209
S_ACT.PGNO2=SDEFAULT.PGNO2
S_ACT.PRESS1=SDEFAULT.PRESS1
S_ACT.PRESS2=SDEFAULT.PRESS2
S_READY=FALSE
PTP XSWP_60_8576
USERSPOT(#SPOT, S_ACT)
WAIT FOR S_READY
;ENDFOLD

;FOLD PTP l171 CONT Vel=100 % fin Tool[4]:Gun C3 Base[3]:Atego/Axor;%{PE}%R 8.2.20,%MKUKATPBASIS,%CMOVE,%VPTP,%P 1:PTP, 2:l171, 3:C_DIS, 5:100, 7:fin
$BWDSTART=FALSE
PDAT_ACT=Pfin
FDAT_ACT=Fl171
BAS(#PTP_PARAMS,100)
PTP Xl171 C_DIS
;ENDFOLD
;FOLD PTP l160 CONT Vel=100 % medium Tool[4]:Gun C3 Base[3]:Atego/Axor;%{PE}%R 8.2.20,%MKUKATPBASIS,%CMOVE,%VPTP,%P 1:PTP, 2:l160, 3:C_DIS, 5:100, 7:medium
$BWDSTART=FALSE
PDAT_ACT=Pmedium
FDAT_ACT=Fl160
BAS(#PTP_PARAMS,100)
PTP Xl160 C_DIS
;ENDFOLD
;FOLD PTP l155 CONT Vel=100 % mediun Tool[4]:Gun C3 Base[3]:Atego/Axor;%{PE}%R 8.2.20,%MKUKATPBASIS,%CMOVE,%VPTP,%P 1:PTP, 2:l155, 3:C_DIS, 5:100, 7:mediun
$BWDSTART=FALSE
PDAT_ACT=Pmediun
FDAT_ACT=Fl155
BAS(#PTP_PARAMS,100)
PTP Xl155 C_DIS
;ENDFOLD
;FOLD PTP l157 CONT Vel=100 % small Tool[4]:Gun C3 Base[3]:Atego/Axor;%{PE}%R 8.2.20,%MKUKATPBASIS,%CMOVE,%VPTP,%P 1:PTP, 2:l157, 3:C_DIS, 5:100, 7:small
$BWDSTART=FALSE
PDAT_ACT=Psmall
FDAT_ACT=Fl157
BAS(#PTP_PARAMS,100)
PTP Xl157 C_DIS
;ENDFOLD
;FOLD PTP l158 CONT Vel=100 % fin Tool[4]:Gun C3 Base[3]:Atego/Axor;%{PE}%R 8.2.20,%MKUKATPBASIS,%CMOVE,%VPTP,%P 1:PTP, 2:l158, 3:C_DIS, 5:100, 7:fin
$BWDSTART=FALSE
PDAT_ACT=Pfin
FDAT_ACT=Fl158
BAS(#PTP_PARAMS,100)
PTP Xl158 C_DIS
;ENDFOLD

;FOLD ; SWP_60_8584;%{PE}%R 8.2.20,%MKUKATPBASIS,%CCOMMENT,%VNORMAL,%P 2:SWP_60_8584
;ENDFOLD
;FOLD PTP SWP_60_8584 vmax SPOT Gun=3 RETR CLS PgNo1=200 ACTIVE=1 Tool[4]:Gun C3 Base[3]:Atego/Axor;%{PE}%R 8.2.2,%MKUKATPSPOT,%CSPOT,%VPTP,%P 1:PTP, 2:SWP_60_8584, 3:, 5:100, 7:vmax, 10:3, 12:#FIRST, 14:#CLO, 16:200, 18:1, 20:0, 22:0, 24:1, 25:NORMAL
$BWDSTART=FALSE
PDAT_ACT=Pvmax
FDAT_ACT=FSWP_60_8584
BAS(#PTP_PARAMS,Pvmax.VEL)
S_ACT.GUN=3
S_ACT.PAIR=SDEFAULT.PAIR
S_ACT.RETR=#CLO
S_ACT.CLO_TM=1
S_ACT.PGNO1=200
S_ACT.PGNO2=SDEFAULT.PGNO2
S_ACT.PRESS1=SDEFAULT.PRESS1
S_ACT.PRESS2=SDEFAULT.PRESS2
S_READY=FALSE
PTP XSWP_60_8584
USERSPOT(#SPOT, S_ACT)
WAIT FOR S_READY
;ENDFOLD

;FOLD ; SWP_60_8788;%{PE}%R 8.2.20,%MKUKATPBASIS,%CCOMMENT,%VNORMAL,%P 2:SWP_60_8788
;ENDFOLD
;FOLD PTP SWP_60_8788 vmax SPOT Gun=3 RETR CLS PgNo1=200 ACTIVE=1 Tool[4]:Gun C3 Base[3]:Atego/Axor;%{PE}%R 8.2.2,%MKUKATPSPOT,%CSPOT,%VPTP,%P 1:PTP, 2:SWP_60_8788, 3:, 5:100, 7:vmax, 10:3, 12:#FIRST, 14:#CLO, 16:200, 18:1, 20:0, 22:0, 24:1, 25:NORMAL
$BWDSTART=FALSE
PDAT_ACT=Pvmax
FDAT_ACT=FSWP_60_8788
BAS(#PTP_PARAMS,Pvmax.VEL)
S_ACT.GUN=3
S_ACT.PAIR=SDEFAULT.PAIR
S_ACT.RETR=#CLO
S_ACT.CLO_TM=1
S_ACT.PGNO1=200
S_ACT.PGNO2=SDEFAULT.PGNO2
S_ACT.PRESS1=SDEFAULT.PRESS1
S_ACT.PRESS2=SDEFAULT.PRESS2
S_READY=FALSE
PTP XSWP_60_8788
USERSPOT(#SPOT, S_ACT)
WAIT FOR S_READY
;ENDFOLD

;FOLD PTP l159 CONT Vel=100 % fin Tool[4]:Gun C3 Base[3]:Atego/Axor;%{PE}%R 8.2.20,%MKUKATPBASIS,%CMOVE,%VPTP,%P 1:PTP, 2:l159, 3:C_DIS, 5:100, 7:fin
$BWDSTART=FALSE
PDAT_ACT=Pfin
FDAT_ACT=Fl159
BAS(#PTP_PARAMS,100)
PTP Xl159 C_DIS
;ENDFOLD
;FOLD PTP l161 CONT Vel=100 % medium Tool[4]:Gun C3 Base[3]:Atego/Axor;%{PE}%R 8.2.20,%MKUKATPBASIS,%CMOVE,%VPTP,%P 1:PTP, 2:l161, 3:C_DIS, 5:100, 7:medium
$BWDSTART=FALSE
PDAT_ACT=Pmedium
FDAT_ACT=Fl161
BAS(#PTP_PARAMS,100)
PTP Xl161 C_DIS
;ENDFOLD
;FOLD PTP l162 CONT Vel=100 % medium Tool[4]:Gun C3 Base[3]:Atego/Axor;%{PE}%R 8.2.20,%MKUKATPBASIS,%CMOVE,%VPTP,%P 1:PTP, 2:l162, 3:C_DIS, 5:100, 7:medium
$BWDSTART=FALSE
PDAT_ACT=Pmedium
FDAT_ACT=Fl162
BAS(#PTP_PARAMS,100)
PTP Xl162 C_DIS
;ENDFOLD
;FOLD PTP l163 CONT Vel=100 % fin Tool[4]:Gun C3 Base[3]:Atego/Axor;%{PE}%R 8.2.20,%MKUKATPBASIS,%CMOVE,%VPTP,%P 1:PTP, 2:l163, 3:C_DIS, 5:100, 7:fin
$BWDSTART=FALSE
PDAT_ACT=Pfin
FDAT_ACT=Fl163
BAS(#PTP_PARAMS,100)
PTP Xl163 C_DIS
;ENDFOLD

;FOLD ; SWP_60_8800;%{PE}%R 8.2.20,%MKUKATPBASIS,%CCOMMENT,%VNORMAL,%P 2:SWP_60_8800
;ENDFOLD
;FOLD PTP SWP_60_8800 vmax SPOT Gun=3 RETR CLS PgNo1=196 ACTIVE=1 Tool[4]:Gun C3 Base[3]:Atego/Axor;%{PE}%R 8.2.2,%MKUKATPSPOT,%CSPOT,%VPTP,%P 1:PTP, 2:SWP_60_8800, 3:, 5:100, 7:vmax, 10:3, 12:#FIRST, 14:#CLO, 16:196, 18:1, 20:0, 22:0, 24:1, 25:NORMAL
$BWDSTART=FALSE
PDAT_ACT=Pvmax
FDAT_ACT=FSWP_60_8800
BAS(#PTP_PARAMS,Pvmax.VEL)
S_ACT.GUN=3
S_ACT.PAIR=SDEFAULT.PAIR
S_ACT.RETR=#CLO
S_ACT.CLO_TM=1
S_ACT.PGNO1=196
S_ACT.PGNO2=SDEFAULT.PGNO2
S_ACT.PRESS1=SDEFAULT.PRESS1
S_ACT.PRESS2=SDEFAULT.PRESS2
S_READY=FALSE
PTP XSWP_60_8800
USERSPOT(#SPOT, S_ACT)
WAIT FOR S_READY
;ENDFOLD

;FOLD PTP l164 CONT Vel=100 % fin Tool[4]:Gun C3 Base[3]:Atego/Axor;%{PE}%R 8.2.20,%MKUKATPBASIS,%CMOVE,%VPTP,%P 1:PTP, 2:l164, 3:C_DIS, 5:100, 7:fin
$BWDSTART=FALSE
PDAT_ACT=Pfin
FDAT_ACT=Fl164
BAS(#PTP_PARAMS,100)
PTP Xl164 C_DIS
;ENDFOLD
;FOLD PTP l166 CONT Vel=100 % small Tool[4]:Gun C3 Base[3]:Atego/Axor;%{PE}%R 8.2.20,%MKUKATPBASIS,%CMOVE,%VPTP,%P 1:PTP, 2:l166, 3:C_DIS, 5:100, 7:small
$BWDSTART=FALSE
PDAT_ACT=Psmall
FDAT_ACT=Fl166
BAS(#PTP_PARAMS,100)
PTP Xl166 C_DIS
;ENDFOLD
;FOLD PTP l150 CONT Vel=100 % small Tool[4]:Gun C3 Base[3]:Atego/Axor;%{PE}%R 8.2.20,%MKUKATPBASIS,%CMOVE,%VPTP,%P 1:PTP, 2:l150, 3:C_DIS, 5:100, 7:small
$BWDSTART=FALSE
PDAT_ACT=Psmall
FDAT_ACT=Fl150
BAS(#PTP_PARAMS,100)
PTP Xl150 C_DIS
;ENDFOLD
;FOLD PTP l145 CONT Vel=100 % small Tool[4]:Gun C3 Base[3]:Atego/Axor;%{PE}%R 8.2.20,%MKUKATPBASIS,%CMOVE,%VPTP,%P 1:PTP, 2:l145, 3:C_DIS, 5:100, 7:small
$BWDSTART=FALSE
PDAT_ACT=Psmall
FDAT_ACT=Fl145
BAS(#PTP_PARAMS,100)
PTP Xl145 C_DIS
;ENDFOLD
;FOLD PTP l135 CONT Vel=100 % fin Tool[4]:Gun C3 Base[3]:Atego/Axor;%{PE}%R 8.2.20,%MKUKATPBASIS,%CMOVE,%VPTP,%P 1:PTP, 2:l135, 3:C_DIS, 5:100, 7:fin
$BWDSTART=FALSE
PDAT_ACT=Pfin
FDAT_ACT=Fl135
BAS(#PTP_PARAMS,100)
PTP Xl135 C_DIS
;ENDFOLD

;FOLD ; SWP_60_8812;%{PE}%R 8.2.20,%MKUKATPBASIS,%CCOMMENT,%VNORMAL,%P 2:SWP_60_8812
;ENDFOLD
;FOLD PTP SWP_60_8812 vmax SPOT Gun=3 RETR OPN PgNo1=207 ACTIVE=1 Tool[4]:Gun C3 Base[3]:Atego/Axor;%{PE}%R 8.2.2,%MKUKATPSPOT,%CSPOT,%VPTP,%P 1:PTP, 2:SWP_60_8812, 3:, 5:100, 7:vmax, 10:3, 12:#FIRST, 14:#OPN, 16:207, 18:1, 20:0, 22:0, 24:1, 25:NORMAL
$BWDSTART=FALSE
PDAT_ACT=Pvmax
FDAT_ACT=FSWP_60_8812
BAS(#PTP_PARAMS,Pvmax.VEL)
S_ACT.GUN=3
S_ACT.PAIR=SDEFAULT.PAIR
S_ACT.RETR=#OPN
S_ACT.CLO_TM=1
S_ACT.PGNO1=207
S_ACT.PGNO2=SDEFAULT.PGNO2
S_ACT.PRESS1=SDEFAULT.PRESS1
S_ACT.PRESS2=SDEFAULT.PRESS2
S_READY=FALSE
PTP XSWP_60_8812
USERSPOT(#SPOT, S_ACT)
WAIT FOR S_READY
;ENDFOLD

;FOLD PTP l130 CONT Vel=100 % fin Tool[4]:Gun C3 Base[3]:Atego/Axor;%{PE}%R 8.2.20,%MKUKATPBASIS,%CMOVE,%VPTP,%P 1:PTP, 2:l130, 3:C_DIS, 5:100, 7:fin
$BWDSTART=FALSE
PDAT_ACT=Pfin
FDAT_ACT=Fl130
BAS(#PTP_PARAMS,100)
PTP Xl130 C_DIS
;ENDFOLD
;FOLD PTP l115 CONT Vel=100 % medium Tool[4]:Gun C3 Base[3]:Atego/Axor;%{PE}%R 8.2.20,%MKUKATPBASIS,%CMOVE,%VPTP,%P 1:PTP, 2:l115, 3:C_DIS, 5:100, 7:medium
$BWDSTART=FALSE
PDAT_ACT=Pmedium
FDAT_ACT=Fl115
BAS(#PTP_PARAMS,100)
PTP Xl115 C_DIS
;ENDFOLD
;FOLD PTP l116 Vel=100 % vmax Tool[4]:Gun C3 Base[3]:Atego/Axor;%{PE}%R 8.2.20,%MKUKATPBASIS,%CMOVE,%VPTP,%P 1:PTP, 2:l116, 3:, 5:100, 7:vmax
$BWDSTART=FALSE
PDAT_ACT=Pvmax
FDAT_ACT=Fl116
BAS(#PTP_PARAMS,100)
PTP Xl116
;ENDFOLD

; FIM DE TRABALHO GEOMETRIA
;FOLD PULSE 3338 'R2 solda geometria Ok' State=TRUE Time=3 sec;%{PE}%R 8.2.20,%MKUKATPBASIS,%COUT,%VPULSE,%P 2:3338, 3:R2 solda geometria Ok, 5:TRUE, 6:, 8:3
PULSE($OUT[3338], TRUE,3)
;ENDFOLD
;FOLD OUT 3348 'Fora area GEOBOX' State=TRUE ;%{PE}%R 8.2.20,%MKUKATPBASIS,%COUT,%VOUTX,%P 2:3348, 3:Fora area GEOBOX, 5:TRUE, 6:
$OUT[3348]=TRUE
;ENDFOLD

; DESLIGA INTERTRAVAMENTO 1 C/ R1
;FOLD Collision.Monitoring_1_Off . ;%{PE}%MKUKATPUSER
COLLSTOP( 1, 2+0 )
;ENDFOLD

; DESLIGA INTERTRAVAMENTO 4 C/ R4
;FOLD Collision.Monitoring_4_Off . ;%{PE}%MKUKATPUSER
COLLSTOP( 4, 2+0 )
;ENDFOLD

; LIGA INTERLOCK 5 C/ R5
;FOLD Collision.Monitoring_5_On ;%{PE}%MKUKATPUSER
COLLSTOP( 5, 1 ) ;not Interrupt-Controlled
;ENDFOLD

;FOLD PTP P6 CONT Vel=100 % xxlarge Tool[4]:Gun C3 Base[3]:Atego/Axor;%{PE}%R 8.2.20,%MKUKATPBASIS,%CMOVE,%VPTP,%P 1:PTP, 2:P6, 3:C_DIS, 5:100, 7:xxlarge
$BWDSTART=FALSE
PDAT_ACT=Pxxlarge
FDAT_ACT=FP6
BAS(#PTP_PARAMS,100)
PTP XP6 C_DIS
;ENDFOLD
;FOLD PTP P3 Vel=100 % vmax Tool[4]:Gun C3 Base[3]:Atego/Axor;%{PE}%R 8.2.20,%MKUKATPBASIS,%CMOVE,%VPTP,%P 1:PTP, 2:P3, 3:, 5:100, 7:vmax
$BWDSTART=FALSE
PDAT_ACT=Pvmax
FDAT_ACT=FP3
BAS(#PTP_PARAMS,100)
PTP XP3
;ENDFOLD

IF (NOT(GHOST())) THEN
if FraesAnf (3) then
 f_fraes4 ()
endif
ENDIF

END

--- ps_b_lta_geo_c03.dat ---
&ACCESS RVO1
&COMMENT Solda Atego LTB
&PARAM DISKPATH = KRC:\R1\Program\OLP
DEFDAT ps_b_lta_geo_c03
;FOLD EXTERNAL DECLARATIONS;%{PE}%MKUKATPBASIS,%CEXT,%VCOMMON,%P
;FOLD GRIPPERTECH EXT
EXT  H50 (INT  :IN,INT  :IN,INT  :IN,GRP_TYP  :IN )
;ENDFOLD (GRIPPERTECH EXT)
;FOLD SPOTTECH EXT
EXT  USERSPOT (S_COMMAND  :IN,SPOT_TYPE  :IN )
;ENDFOLD (SPOTTECH EXT)
;FOLD BASISTECH EXT;%{PE}%MKUKATPBASIS,%CEXT,%VEXT,%P
EXT  BAS (BAS_COMMAND  :IN,REAL  :IN )
DECL INT SUCCESS
;ENDFOLD (BASISTECH EXT)
;FOLD USER EXT;%{E}%MKUKATPUSER,%CEXT,%VEXT,%P
;Make your modifications here

;ENDFOLD (USER EXT)
;ENDFOLD (EXTERNAL DECLARATIONS)



DECL PDAT PP_OLP4={VEL 100.0,ACC 100.0,APO_DIST 20.0,APO_MODE #CDIS}
DECL PDAT PP_OLP7={VEL 100.0,ACC 100.0,APO_DIST 100.0,APO_MODE #CDIS}


; E6POS declarations
; FDAT declarations
; LDAT declarations
; PDAT declarations

; E6POS declarations
DECL E6POS XSWP_60_9078={X 377.429504,Y 998.692078,Z -51.6705818,A -178.750397,B 54.3092003,C 89.6855087,S 2,T 11,E1 -5500.00195,E2 0.0,E3 0.0,E4 0.0,E5 0.0,E6 0.0}
DECL E6POS XSWP_60_8584={X 574.901672,Y 959.645203,Z 1312.65002,A -171.738693,B -53.4007301,C 82.1439133,S 2,T 11,E1 -5500.0,E2 0.0,E3 0.0,E4 0.0,E5 0.0,E6 0.0}
DECL E6POS XSWP_60_8788={X 685.193909,Y 955.620117,Z 1322.33398,A -124.007103,B -84.2773209,C 35.6398811,S 2,T 11,E1 -5500.0,E2 0.0,E3 0.0,E4 0.0,E5 0.0,E6 0.0}
DECL E6POS XSWP_60_8800={X 959.385071,Y 969.231201,Z 1333.18396,A -9.99958229,B -68.941597,C -77.7464828,S 2,T 11,E1 -5500.0,E2 0.0,E3 0.0,E4 0.0,E5 0.0,E6 0.0}
DECL E6POS Xl115={X 1235.03198,Y 1367.06604,Z 1292.71497,A -80.0313873,B -85.9020309,C -9.10745239,S 2,T 10,E1 -5500.0,E2 0.0,E3 0.0,E4 0.0,E5 0.0,E6 0.0}
DECL E6POS Xl130={X 1231.23999,Y 962.339111,Z 1297.51001,A -81.1379089,B -84.6478424,C -7.77770805,S 2,T 11,E1 -5499.99902,E2 0.0,E3 0.0,E4 0.0,E5 0.0,E6 0.0}
DECL E6POS XSWP_60_8812={X 1232.76001,Y 973.570801,Z 1334.12903,A -79.7475128,B -85.9006195,C -9.10391426,S 2,T 11,E1 -5499.99902,E2 0.0,E3 0.0,E4 0.0,E5 0.0,E6 0.0}
DECL E6POS Xl135={X 1231.23999,Y 962.339111,Z 1297.51001,A -81.1379089,B -84.6478424,C -7.77770805,S 2,T 11,E1 -5499.99902,E2 0.0,E3 0.0,E4 0.0,E5 0.0,E6 0.0}
DECL E6POS Xl145={X 1225.06006,Y 1267.27502,Z 1289.97595,A -82.990799,B -85.3915329,C -5.86582804,S 2,T 10,E1 -5500.0,E2 0.0,E3 0.0,E4 0.0,E5 0.0,E6 0.0}
DECL E6POS Xl150={X 1084.92798,Y 1289.59802,Z 1316.64697,A -110.132202,B -85.2466202,C 21.2871304,S 2,T 10,E1 -5500.0,E2 0.0,E3 0.0,E4 0.0,E5 0.0,E6 0.0}
DECL E6POS Xl155={X 495.042297,Y 1192.729,Z 1176.08704,A -166.6194,B -62.0061798,C 77.3858871,S 2,T 10,E1 -5500.0,E2 0.0,E3 0.0,E4 0.0,E5 0.0,E6 0.0}
DECL E6POS Xl160={X 495.625793,Y 1048.98596,Z 1173.58606,A -166.463699,B -59.9506111,C 75.8885117,S 2,T 11,E1 -5500.0,E2 0.0,E3 0.0,E4 0.0,E5 0.0,E6 0.0}
DECL E6POS XSWP_60_8576={X 479.7323,Y 961.704895,Z 1232.96802,A -168.522095,B -65.2164001,C 79.4213181,S 2,T 11,E1 -5500.0,E2 0.0,E3 0.0,E4 0.0,E5 0.0,E6 0.0}
DECL E6POS Xl170={X 493.426605,Y 954.01123,Z 1196.677,A -165.408203,B -64.9694595,C 76.488472,S 2,T 11,E1 -5500.0,E2 0.0,E3 0.0,E4 0.0,E5 0.0,E6 0.0}
DECL E6POS Xl175={X 498.414612,Y 1048.99402,Z 1175.27905,A -167.799103,B -56.2781601,C 76.6106262,S 2,T 11,E1 -5500.0,E2 0.0,E3 0.0,E4 0.0,E5 0.0,E6 0.0}
DECL E6POS Xl180={X 504.707489,Y 1257.96997,Z 1171.14404,A -175.011902,B -65.2939529,C 85.5748062,S 2,T 10,E1 -5500.0,E2 0.0,E3 0.0,E4 0.0,E5 0.0,E6 0.0}
DECL E6POS Xl185={X 281.523285,Y 1267.26001,Z -80.7737808,A -171.102203,B -55.8212395,C 78.1676636,S 2,T 10,E1 -5500.00195,E2 0.0,E3 0.0,E4 0.0,E5 0.0,E6 0.0}
DECL E6POS Xl195={X 309.236694,Y 1189.24902,Z -261.055695,A -161.565903,B -64.5644531,C 71.0960388,S 2,T 10,E1 -5500.00586,E2 0.0,E3 0.0,E4 0.0,E5 0.0,E6 0.0}
DECL E6POS Xl200={X 320.765808,Y 952.112915,Z -276.100006,A -170.774399,B -65.5663605,C 82.4341507,S 2,T 11,E1 -5500.00586,E2 0.0,E3 0.0,E4 0.0,E5 0.0,E6 0.0}
DECL E6POS XSWP_60_8046={X 295.258392,Y 953.246582,Z -191.709198,A -178.112198,B -65.694397,C 89.5197296,S 2,T 11,E1 -5500.00586,E2 0.0,E3 0.0,E4 0.0,E5 0.0,E6 0.0}
DECL E6POS Xl205={X 313.821808,Y 939.276306,Z -206.506302,A -176.364502,B -65.6938019,C 88.284462,S 2,T 11,E1 -5500.00586,E2 0.0,E3 0.0,E4 0.0,E5 0.0,E6 0.0}
DECL E6POS Xl210={X 320.765808,Y 952.112915,Z -276.100006,A -170.774399,B -65.5663528,C 82.4341507,S 2,T 11,E1 -5500.00586,E2 0.0,E3 0.0,E4 0.0,E5 0.0,E6 0.0}
DECL E6POS Xl215={X 311.768311,Y 1138.82202,Z -260.171997,A -172.248505,B -65.4501114,C 83.7742386,S 2,T 10,E1 -5500.00586,E2 0.0,E3 0.0,E4 0.0,E5 0.0,E6 0.0}
DECL E6POS Xl220={X 321.698212,Y 1495.271,Z -235.324005,A 177.775497,B -76.9053802,C 89.1578827,S 2,T 10,E1 -5500.0,E2 0.0,E3 0.0,E4 0.0,E5 0.0,E6 0.0}
DECL E6POS Xl225={X 511.616211,Y 1495.66797,Z -217.2724,A -176.421494,B -85.6921997,C 87.4376068,S 2,T 10,E1 -5500.0,E2 0.0,E3 0.0,E4 0.0,E5 0.0,E6 0.0}
DECL E6POS Xl230={X 561.25293,Y 949.928406,Z -209.439102,A -162.895203,B -85.5735092,C 75.3529587,S 2,T 11,E1 -5499.99805,E2 0.0,E3 0.0,E4 0.0,E5 0.0,E6 0.0}
DECL E6POS XSWP_60_8060={X 512.477783,Y 955.514282,Z -183.049194,A -176.456406,B -85.6937866,C 87.4698563,S 2,T 11,E1 -5499.99805,E2 0.0,E3 0.0,E4 0.0,E5 0.0,E6 0.0}
DECL E6POS Xl240={X 561.25293,Y 949.928406,Z -209.439102,A -162.895203,B -85.5735092,C 75.3529587,S 2,T 11,E1 -5499.99805,E2 0.0,E3 0.0,E4 0.0,E5 0.0,E6 0.0}
DECL E6POS Xl250={X 534.108521,Y 1051.99402,Z -234.229004,A -178.033707,B -27.6022606,C 88.6840973,S 2,T 11,E1 -5500.0,E2 0.0,E3 0.0,E4 0.0,E5 0.0,E6 0.0}
DECL E6POS Xl255={X 526.619873,Y 1071.71301,Z -83.3147964,A -178.809601,B 34.4082718,C 89.7623367,S 2,T 10,E1 -5500.0,E2 0.0,E3 0.0,E4 0.0,E5 0.0,E6 0.0}
DECL E6POS Xl265={X 552.832581,Y 992.614319,Z -76.7540436,A -177.865707,B 43.6499786,C 90.5385971,S 2,T 11,E1 -5500.00488,E2 0.0,E3 0.0,E4 0.0,E5 0.0,E6 0.0}
DECL E6POS XSWP_60_8068={X 522.917725,Y 999.467896,Z -110.008202,A -178.878799,B 43.6501999,C 89.7160492,S 2,T 11,E1 -5500.00488,E2 0.0,E3 0.0,E4 0.0,E5 0.0,E6 0.0}
DECL E6POS Xl270={X 552.832581,Y 992.614319,Z -76.7540436,A -177.865707,B 43.6499786,C 90.5385971,S 2,T 11,E1 -5500.00488,E2 0.0,E3 0.0,E4 0.0,E5 0.0,E6 0.0}
DECL E6POS Xl280={X 675.09613,Y 1281.73804,Z -58.8733101,A 178.420898,B 65.5474091,C 89.3197327,S 2,T 10,E1 -5500.0,E2 0.0,E3 0.0,E4 0.0,E5 0.0,E6 0.0}
DECL E6POS Xl285={X 1138.53101,Y 1467.13,Z 160.281296,A -5.84426117,B 62.4796715,C -83.9085999,S 2,T 42,E1 -4299.99609,E2 0.0,E3 0.0,E4 0.0,E5 0.0,E6 0.0}
DECL E6POS Xl290={X 1258.77795,Y 1189.58606,Z 206.930603,A -3.86018109,B 62.4975014,C -87.444603,S 2,T 42,E1 -4299.99609,E2 0.0,E3 0.0,E4 0.0,E5 0.0,E6 0.0}
DECL E6POS Xl295={X 1235.88,Y 988.000793,Z 245.895401,A -4.5130868,B 55.8284912,C -88.7858887,S 2,T 43,E1 -4299.99609,E2 0.0,E3 0.0,E4 0.0,E5 0.0,E6 0.0}
DECL E6POS XSWP_60_8542={X 1267.56702,Y 1004.06097,Z 212.281006,A -1.81140697,B 56.6370506,C -86.7754364,S 2,T 43,E1 -4299.99609,E2 0.0,E3 0.0,E4 0.0,E5 0.0,E6 0.0}
DECL E6POS Xl300={X 1235.88,Y 988.000793,Z 245.895401,A -4.5130868,B 55.8284912,C -88.7858887,S 2,T 43,E1 -4299.99609,E2 0.0,E3 0.0,E4 0.0,E5 0.0,E6 0.0}
DECL E6POS Xl310={X 1258.77795,Y 1189.58606,Z 206.930603,A -3.86018109,B 62.4975014,C -87.444603,S 2,T 42,E1 -4299.99609,E2 0.0,E3 0.0,E4 0.0,E5 0.0,E6 0.0}
DECL E6POS Xl320={X 1352.18506,Y 1242.99304,Z 206.460297,A 15.1004696,B 86.7669067,C -72.9232407,S 2,T 42,E1 -4300.00488,E2 0.0,E3 0.0,E4 0.0,E5 0.0,E6 0.0}
DECL E6POS Xl325={X 1360.85901,Y 997.07312,Z 389.614502,A -5.78831482,B 64.6253586,C -93.8561096,S 2,T 43,E1 -4300.00391,E2 0.0,E3 0.0,E4 0.0,E5 0.0,E6 0.0}
DECL E6POS XSWP_60_8554={X 1389.12695,Y 1005.08197,Z 361.854797,A -2.05229092,B 49.6726303,C -91.4522171,S 2,T 43,E1 -4300.00391,E2 0.0,E3 0.0,E4 0.0,E5 0.0,E6 0.0}
DECL E6POS Xl330={X 1362.09302,Y 991.111877,Z 390.607513,A -4.98367405,B 58.5645905,C -93.3877182,S 2,T 43,E1 -4300.00391,E2 0.0,E3 0.0,E4 0.0,E5 0.0,E6 0.0}
DECL E6POS Xl335={X 1373.38904,Y 1246.448,Z 357.980988,A -174.020905,B 79.9130096,C 97.8761673,S 2,T 42,E1 -4300.00488,E2 0.0,E3 0.0,E4 0.0,E5 0.0,E6 0.0}
DECL E6POS Xl350={X 1384.01501,Y 1252.80298,Z 90.7271194,A -176.196106,B -35.5967903,C 87.3916931,S 2,T 10,E1 -4300.01123,E2 0.0,E3 0.0,E4 0.0,E5 0.0,E6 0.0}
DECL E6POS Xl355={X 1332.70496,Y 1026.69397,Z 64.0089569,A -169.138702,B -75.4985504,C 80.5394363,S 2,T 11,E1 -4300.01123,E2 0.0,E3 0.0,E4 0.0,E5 0.0,E6 0.0}
DECL E6POS XSWP_60_8534={X 1304.84802,Y 1022.612,Z 128.3629,A -178.765793,B -75.696991,C 89.4786072,S 2,T 11,E1 -4300.01123,E2 0.0,E3 0.0,E4 0.0,E5 0.0,E6 0.0}
DECL E6POS XSWP_60_8526={X 1475.323,Y 1022.42401,Z 136.200302,A -176.310898,B -87.5757828,C 85.9231567,S 2,T 11,E1 -4300.03223,E2 0.0,E3 0.0,E4 0.0,E5 0.0,E6 0.0}
DECL E6POS XSWP_60_8518={X 1617.62,Y 1021.716,Z 138.371796,A -162.126404,B -89.4310837,C 71.7452698,S 2,T 11,E1 -4300.04297,E2 0.0,E3 0.0,E4 0.0,E5 0.0,E6 0.0}
DECL E6POS Xl380={X 1784.21106,Y 1015.104,Z 120.173203,A -172.612305,B -82.3815765,C 83.4273376,S 2,T 11,E1 -4300.0459,E2 0.0,E3 0.0,E4 0.0,E5 0.0,E6 0.0}
DECL E6POS XSWP_60_8506={X 1906.48999,Y 1020.21899,Z 136.589706,A -178.820999,B -75.6970673,C 89.2493286,S 2,T 11,E1 -4300.04883,E2 0.0,E3 0.0,E4 0.0,E5 0.0,E6 0.0}
DECL E6POS XSWP_60_8494={X 2205.76001,Y 1021.89899,Z 136.038498,A -177.086899,B -85.6936722,C 87.530777,S 2,T 11,E1 -4300.04199,E2 0.0,E3 0.0,E4 0.0,E5 0.0,E6 0.0}
DECL E6POS Xl385={X 2194.77588,Y 1008.60303,Z 109.026497,A -165.4086,B -85.5601196,C 75.4293137,S 2,T 11,E1 -4300.04102,E2 0.0,E3 0.0,E4 0.0,E5 0.0,E6 0.0}
DECL E6POS Xl390={X 2063.57593,Y 1158.78003,Z -1.02906096,A -113.352203,B -73.1949387,C 20.2263699,S 2,T 10,E1 -4300.04102,E2 0.0,E3 0.0,E4 0.0,E5 0.0,E6 0.0}
DECL E6POS Xl395={X 2274.67407,Y 1433.00598,Z 32.1655388,A -83.3964081,B -47.8502388,C -5.32451487,S 2,T 11,E1 -4300.03516,E2 0.0,E3 0.0,E4 0.0,E5 0.0,E6 0.0}
DECL E6POS Xl400={X 2454.4939,Y 1423.14197,Z -2.76967096,A -93.6481018,B -35.0793495,C 2.75330591,S 2,T 11,E1 -4300.03223,E2 0.0,E3 0.0,E4 0.0,E5 0.0,E6 0.0}
DECL E6POS Xl405={X 2842.94092,Y 1365.24597,Z -80.7003632,A -106.436302,B -21.1004696,C 6.97002316,S 2,T 11,E1 -4300.02393,E2 0.0,E3 0.0,E4 0.0,E5 0.0,E6 0.0}
DECL E6POS Xl410={X 2950.46509,Y 1243.85999,Z -185.898499,A -126.371597,B -19.8252792,C 0.398173302,S 2,T 3,E1 -4300.0332,E2 0.0,E3 0.0,E4 0.0,E5 0.0,E6 0.0}
DECL E6POS Xl415={X 2696.40796,Y 517.301208,Z -189.411102,A -139.132706,B -44.6192398,C -12.8349895,S 2,T 35,E1 -4299.99805,E2 0.0,E3 0.0,E4 0.0,E5 0.0,E6 0.0}
DECL E6POS Xl420={X 2236.91089,Y 136.768997,Z 305.577301,A 93.3859024,B -75.1966934,C 86.5297623,S 2,T 35,E1 -4300.01807,E2 0.0,E3 0.0,E4 0.0,E5 0.0,E6 0.0}
DECL E6POS XSWP_60_9462={X 2235.64404,Y 124.546402,Z 351.346802,A 87.8143463,B -75.1700363,C 92.7289581,S 2,T 35,E1 -4300.01807,E2 0.0,E3 0.0,E4 0.0,E5 0.0,E6 0.0}
DECL E6POS XSWP_60_9472={X 2239.97412,Y 354.103302,Z 274.737915,A 88.9424591,B -65.1767807,C 91.6637268,S 2,T 35,E1 -4300.0498,E2 0.0,E3 0.0,E4 0.0,E5 0.0,E6 0.0}
DECL E6POS Xl450={X 2230.72192,Y 324.583099,Z 253.623398,A 91.534523,B -65.1934433,C 89.9227829,S 2,T 35,E1 -4300.0498,E2 0.0,E3 0.0,E4 0.0,E5 0.0,E6 0.0}
DECL E6POS Xl460={X 2345.0791,Y 285.238007,Z 206.417404,A 94.2857437,B -68.3308563,C 89.9274368,S 2,T 35,E1 -4300.0498,E2 0.0,E3 0.0,E4 0.0,E5 0.0,E6 0.0}
DECL E6POS Xl465={X 2355.8501,Y 591.258484,Z 85.2902985,A -95.9454269,B -83.3990936,C -81.5240326,S 2,T 35,E1 -4300.04004,E2 0.0,E3 0.0,E4 0.0,E5 0.0,E6 0.0}
DECL E6POS Xl470={X 2233.84009,Y 688.028625,Z 86.8898163,A -94.4168167,B -74.736412,C -86.3317184,S 2,T 35,E1 -4300.04004,E2 0.0,E3 0.0,E4 0.0,E5 0.0,E6 0.0}
DECL E6POS XSWP_60_9476={X 2240.552,Y 649.875122,Z 135.006302,A -86.9652328,B -74.8011627,C -92.6756897,S 2,T 35,E1 -4300.04004,E2 0.0,E3 0.0,E4 0.0,E5 0.0,E6 0.0}
DECL E6POS Xl475={X 2232.521,Y 659.59613,Z 110.005302,A -90.4983673,B -74.8003235,C -89.3733597,S 2,T 35,E1 -4300.04004,E2 0.0,E3 0.0,E4 0.0,E5 0.0,E6 0.0}
DECL E6POS Xl480={X 2257.198,Y 886.101929,Z -170.302307,A -110.028999,B -67.609108,C -75.7798462,S 2,T 35,E1 -4300.04004,E2 0.0,E3 0.0,E4 0.0,E5 0.0,E6 0.0}
DECL E6POS Xl490={X 2384.25708,Y 1012.56799,Z -192.055405,A -173.582993,B -79.7526169,C -5.49809599,S 2,T 35,E1 -4299.98291,E2 0.0,E3 0.0,E4 0.0,E5 0.0,E6 0.0}
DECL E6POS Xl495={X 2232.46899,Y 1000.383,Z 113.206497,A 93.009903,B -85.2273636,C 87.7077789,S 2,T 35,E1 -4300.00293,E2 0.0,E3 0.0,E4 0.0,E5 0.0,E6 0.0}
DECL E6POS XSWP_60_9492={X 2242.71802,Y 1006.38202,Z 135.158997,A 83.7456894,B -85.1959686,C 96.8084869,S 2,T 35,E1 -4300.00293,E2 0.0,E3 0.0,E4 0.0,E5 0.0,E6 0.0}
DECL E6POS Xl500={X 2232.46899,Y 1000.383,Z 113.206497,A 93.009903,B -85.2273636,C 87.7077789,S 2,T 35,E1 -4300.00293,E2 0.0,E3 0.0,E4 0.0,E5 0.0,E6 0.0}
DECL E6POS Xl505={X 2374.02905,Y 1009.883,Z -131.8918,A -174.716202,B -81.7690735,C -4.57352781,S 2,T 35,E1 -4299.98291,E2 0.0,E3 0.0,E4 0.0,E5 0.0,E6 0.0}
DECL E6POS Xl515={X 2605.12988,Y 695.409912,Z -233.345093,A -155.662704,B -50.6982002,C -24.0847492,S 2,T 35,E1 -4300.0,E2 0.0,E3 0.0,E4 0.0,E5 0.0,E6 0.0}
DECL E6POS Xl520={X 2898.14502,Y 788.585083,Z -372.326813,A -171.528503,B -35.557621,C 4.93190002,S 2,T 35,E1 -4300.01416,E2 0.0,E3 0.0,E4 0.0,E5 0.0,E6 0.0}
; FDAT declarations
DECL FDAT FSWP_60_9078={TOOL_NO 4,BASE_NO 3,IPO_FRAME #BASE,POINT2[] " "}
DECL FDAT FSWP_60_8584={TOOL_NO 4,BASE_NO 3,IPO_FRAME #BASE,POINT2[] " ",TQ_STATE FALSE}
DECL FDAT FSWP_60_8788={TOOL_NO 4,BASE_NO 3,IPO_FRAME #BASE,POINT2[] " "}
DECL FDAT FSWP_60_8800={TOOL_NO 4,BASE_NO 3,IPO_FRAME #BASE,POINT2[] " "}
DECL FDAT Fl115={TOOL_NO 4,BASE_NO 3,IPO_FRAME #BASE,POINT2[] " "}
DECL FDAT Fl130={TOOL_NO 4,BASE_NO 3,IPO_FRAME #BASE,POINT2[] " "}
DECL FDAT FSWP_60_8812={TOOL_NO 4,BASE_NO 3,IPO_FRAME #BASE,POINT2[] " "}
DECL FDAT Fl135={TOOL_NO 4,BASE_NO 3,IPO_FRAME #BASE,POINT2[] " "}
DECL FDAT Fl145={TOOL_NO 4,BASE_NO 3,IPO_FRAME #BASE,POINT2[] " "}
DECL FDAT Fl150={TOOL_NO 4,BASE_NO 3,IPO_FRAME #BASE,POINT2[] " "}
DECL FDAT Fl155={TOOL_NO 4,BASE_NO 3,IPO_FRAME #BASE,POINT2[] " "}
DECL FDAT Fl160={TOOL_NO 4,BASE_NO 3,IPO_FRAME #BASE,POINT2[] " "}
DECL FDAT FSWP_60_8576={TOOL_NO 4,BASE_NO 3,IPO_FRAME #BASE,POINT2[] " "}
DECL FDAT Fl170={TOOL_NO 4,BASE_NO 3,IPO_FRAME #BASE,POINT2[] " "}
DECL FDAT Fl175={TOOL_NO 4,BASE_NO 3,IPO_FRAME #BASE,POINT2[] " "}
DECL FDAT Fl180={TOOL_NO 4,BASE_NO 3,IPO_FRAME #BASE,POINT2[] " "}
DECL FDAT Fl185={TOOL_NO 4,BASE_NO 3,IPO_FRAME #BASE,POINT2[] " "}
DECL FDAT Fl195={TOOL_NO 4,BASE_NO 3,IPO_FRAME #BASE,POINT2[] " "}
DECL FDAT Fl200={TOOL_NO 4,BASE_NO 3,IPO_FRAME #BASE,POINT2[] " "}
DECL FDAT FSWP_60_8046={TOOL_NO 4,BASE_NO 3,IPO_FRAME #BASE,POINT2[] " "}
DECL FDAT Fl205={TOOL_NO 4,BASE_NO 3,IPO_FRAME #BASE,POINT2[] " "}
DECL FDAT Fl210={TOOL_NO 4,BASE_NO 3,IPO_FRAME #BASE,POINT2[] " "}
DECL FDAT Fl215={TOOL_NO 4,BASE_NO 3,IPO_FRAME #BASE,POINT2[] " "}
DECL FDAT Fl220={TOOL_NO 4,BASE_NO 3,IPO_FRAME #BASE,POINT2[] " "}
DECL FDAT Fl225={TOOL_NO 4,BASE_NO 3,IPO_FRAME #BASE,POINT2[] " "}
DECL FDAT Fl230={TOOL_NO 4,BASE_NO 3,IPO_FRAME #BASE,POINT2[] " "}
DECL FDAT FSWP_60_8060={TOOL_NO 4,BASE_NO 3,IPO_FRAME #BASE,POINT2[] " "}
DECL FDAT Fl240={TOOL_NO 4,BASE_NO 3,IPO_FRAME #BASE,POINT2[] " "}
DECL FDAT Fl250={TOOL_NO 4,BASE_NO 3,IPO_FRAME #BASE,POINT2[] " "}
DECL FDAT Fl255={TOOL_NO 4,BASE_NO 3,IPO_FRAME #BASE,POINT2[] " "}
DECL FDAT Fl265={TOOL_NO 4,BASE_NO 3,IPO_FRAME #BASE,POINT2[] " "}
DECL FDAT FSWP_60_8068={TOOL_NO 4,BASE_NO 3,IPO_FRAME #BASE,POINT2[] " "}
DECL FDAT Fl270={TOOL_NO 4,BASE_NO 3,IPO_FRAME #BASE,POINT2[] " "}
DECL FDAT Fl280={TOOL_NO 4,BASE_NO 3,IPO_FRAME #BASE,POINT2[] " "}
DECL FDAT Fl285={TOOL_NO 4,BASE_NO 3,IPO_FRAME #BASE,POINT2[] " "}
DECL FDAT Fl290={TOOL_NO 4,BASE_NO 3,IPO_FRAME #BASE,POINT2[] " "}
DECL FDAT Fl295={TOOL_NO 4,BASE_NO 3,IPO_FRAME #BASE,POINT2[] " "}
DECL FDAT FSWP_60_8542={TOOL_NO 4,BASE_NO 3,IPO_FRAME #BASE,POINT2[] " "}
DECL FDAT Fl300={TOOL_NO 4,BASE_NO 3,IPO_FRAME #BASE,POINT2[] " "}
DECL FDAT Fl310={TOOL_NO 4,BASE_NO 3,IPO_FRAME #BASE,POINT2[] " "}
DECL FDAT Fl320={TOOL_NO 4,BASE_NO 3,IPO_FRAME #BASE,POINT2[] " "}
DECL FDAT Fl325={TOOL_NO 4,BASE_NO 3,IPO_FRAME #BASE,POINT2[] " "}
DECL FDAT FSWP_60_8554={TOOL_NO 4,BASE_NO 3,IPO_FRAME #BASE,POINT2[] " "}
DECL FDAT Fl330={TOOL_NO 4,BASE_NO 3,IPO_FRAME #BASE,POINT2[] " "}
DECL FDAT Fl335={TOOL_NO 4,BASE_NO 3,IPO_FRAME #BASE,POINT2[] " "}
DECL FDAT Fl350={TOOL_NO 4,BASE_NO 3,IPO_FRAME #BASE,POINT2[] " "}
DECL FDAT Fl355={TOOL_NO 4,BASE_NO 3,IPO_FRAME #BASE,POINT2[] " "}
DECL FDAT FSWP_60_8534={TOOL_NO 4,BASE_NO 3,IPO_FRAME #BASE,POINT2[] " "}
DECL FDAT FSWP_60_8526={TOOL_NO 4,BASE_NO 3,IPO_FRAME #BASE,POINT2[] " "}
DECL FDAT FSWP_60_8518={TOOL_NO 4,BASE_NO 3,IPO_FRAME #BASE,POINT2[] " "}
DECL FDAT Fl380={TOOL_NO 4,BASE_NO 3,IPO_FRAME #BASE,POINT2[] " "}
DECL FDAT FSWP_60_8506={TOOL_NO 4,BASE_NO 3,IPO_FRAME #BASE,POINT2[] " "}
DECL FDAT FSWP_60_8494={TOOL_NO 4,BASE_NO 3,IPO_FRAME #BASE,POINT2[] " "}
DECL FDAT Fl385={TOOL_NO 4,BASE_NO 3,IPO_FRAME #BASE,POINT2[] " "}
DECL FDAT Fl390={TOOL_NO 4,BASE_NO 3,IPO_FRAME #BASE,POINT2[] " "}
DECL FDAT Fl395={TOOL_NO 4,BASE_NO 3,IPO_FRAME #BASE,POINT2[] " "}
DECL FDAT Fl400={TOOL_NO 4,BASE_NO 3,IPO_FRAME #BASE,POINT2[] " "}
DECL FDAT Fl405={TOOL_NO 4,BASE_NO 3,IPO_FRAME #BASE,POINT2[] " "}
DECL FDAT Fl410={TOOL_NO 4,BASE_NO 3,IPO_FRAME #BASE,POINT2[] " "}
DECL FDAT Fl415={TOOL_NO 4,BASE_NO 3,IPO_FRAME #BASE,POINT2[] " "}
DECL FDAT Fl420={TOOL_NO 4,BASE_NO 3,IPO_FRAME #BASE,POINT2[] " "}
DECL FDAT FSWP_60_9462={TOOL_NO 4,BASE_NO 3,IPO_FRAME #BASE,POINT2[] " "}
DECL FDAT FSWP_60_9472={TOOL_NO 4,BASE_NO 3,IPO_FRAME #BASE,POINT2[] " "}
DECL FDAT Fl450={TOOL_NO 4,BASE_NO 3,IPO_FRAME #BASE,POINT2[] " "}
DECL FDAT Fl460={TOOL_NO 4,BASE_NO 3,IPO_FRAME #BASE,POINT2[] " "}
DECL FDAT Fl465={TOOL_NO 4,BASE_NO 3,IPO_FRAME #BASE,POINT2[] " "}
DECL FDAT Fl470={TOOL_NO 4,BASE_NO 3,IPO_FRAME #BASE,POINT2[] " "}
DECL FDAT FSWP_60_9476={TOOL_NO 4,BASE_NO 3,IPO_FRAME #BASE,POINT2[] " "}
DECL FDAT Fl475={TOOL_NO 4,BASE_NO 3,IPO_FRAME #BASE,POINT2[] " "}
DECL FDAT Fl480={TOOL_NO 4,BASE_NO 3,IPO_FRAME #BASE,POINT2[] " "}
DECL FDAT Fl490={TOOL_NO 4,BASE_NO 3,IPO_FRAME #BASE,POINT2[] " "}
DECL FDAT Fl495={TOOL_NO 4,BASE_NO 3,IPO_FRAME #BASE,POINT2[] " "}
DECL FDAT FSWP_60_9492={TOOL_NO 4,BASE_NO 3,IPO_FRAME #BASE,POINT2[] " "}
DECL FDAT Fl500={TOOL_NO 4,BASE_NO 3,IPO_FRAME #BASE,POINT2[] " "}
DECL FDAT Fl505={TOOL_NO 4,BASE_NO 3,IPO_FRAME #BASE,POINT2[] " "}
DECL FDAT Fl515={TOOL_NO 4,BASE_NO 3,IPO_FRAME #BASE,POINT2[] " "}
DECL FDAT Fl520={TOOL_NO 4,BASE_NO 3,IPO_FRAME #BASE,POINT2[] " "}
; LDAT declarations
; PDAT declarations
DECL PDAT PP_OLP48={VEL 100.0,ACC 100.0,APO_DIST 100.0,APO_MODE #CDIS}

DECL BASIS_SUGG_T LAST_BASIS={POINT1[] "P0                      ",POINT2[] "P0                      ",CP_PARAMS[] "CPDAT0                  ",PTP_PARAMS[] "PDAT0                   ",CONT[] "                        ",CP_VEL[] "2.0                     ",PTP_VEL[] " 100                    ",SYNC_PARAMS[] "SYNCDAT                 ",SPL_NAME[] "S0                      "}
DECL E6POS XP3={X 6613.13721,Y 2724.13306,Z -373.286285,A 177.972305,B -19.9949894,C 0.623903513,S 2,T 10,E1 199.999695,E2 0.0,E3 0.0,E4 0.0,E5 0.0,E6 0.0}
DECL FDAT FP3={TOOL_NO 4,BASE_NO 3,IPO_FRAME #BASE,POINT2[] " ",TQ_STATE FALSE}
DECL E6POS XP4={X 6609.03711,Y 2724.14111,Z -373.300293,A 177.973007,B -20.0004101,C 0.623480797,S 2,T 2,E1 450.927094,E2 0.0,E3 0.0,E4 0.0,E5 0.0,E6 0.0}
DECL FDAT FP4={TOOL_NO 4,BASE_NO 3,IPO_FRAME #BASE,POINT2[] " ",TQ_STATE FALSE}
DECL PDAT PPDAT5={VEL 100.0,ACC 100.0,APO_DIST 100.0,APO_MODE #CDIS}
DECL PDAT PP_OLP71={VEL 100.0,ACC 100.0,APO_DIST 100.0,APO_MODE #CDIS}
DECL E6POS Xl526={X 3354.73999,Y 2478.89404,Z 10.7530003,A -163.420303,B -21.2028999,C -0.973699987,S 2,T 11,E1 -3400.0,E2 0.0,E3 0.0,E4 0.0,E5 0.0,E6 0.0}
DECL FDAT Fl526={TOOL_NO 4,BASE_NO 3,IPO_FRAME #BASE,POINT2[] " "}
DECL E6POS XP5={X 2041.26001,Y 1013.46198,Z 123.198303,A -175.309402,B -79.8184433,C 86.2517471,S 2,T 11,E1 -4300.0459,E2 0.0,E3 0.0,E4 0.0,E5 0.0,E6 0.0}
DECL FDAT FP5={TOOL_NO 4,BASE_NO 3,IPO_FRAME #BASE,POINT2[] " ",TQ_STATE FALSE}
DECL SPOT_SUGG_T LAST_SPOT={GUN[] "1                       ",RETR_CMD[] "#OPN                    ",CHOISE[] "#FIRST                  ",CLO_TM[] "0                       ",PGNO1[] "1                       ",PRESS1[] "0                       ",PGNO2[] "1                       ",PRESS2[] "0                       ",SPOT_PARAMS[] "NORMAL                  "}
DECL E6POS XP6={X 4327.83887,Y 2781.13696,Z 101.617104,A -125.010002,B -30.4753895,C -36.3488693,S 2,T 10,E1 -1429.17603,E2 0.0,E3 0.0,E4 0.0,E5 0.0,E6 0.0}
DECL FDAT FP6={TOOL_NO 4,BASE_NO 3,IPO_FRAME #BASE,POINT2[] " ",TQ_STATE FALSE}
DECL E6POS Xl186={X 375.888885,Y 1351.16699,Z 785.390381,A 179.603394,B -35.7009315,C 85.0550385,S 2,T 10,E1 -5500.0,E2 0.0,E3 0.0,E4 0.0,E5 0.0,E6 0.0}
DECL FDAT Fl186={TOOL_NO 4,BASE_NO 3,IPO_FRAME #BASE,POINT2[] " "}
DECL E6POS Xl107={X 2242.42505,Y 256.580109,Z 231.991699,A 95.0900269,B -66.7449265,C 87.0306091,S 2,T 35,E1 -4300.04492,E2 0.0,E3 0.0,E4 0.0,E5 0.0,E6 0.0}
DECL FDAT Fl107={TOOL_NO 4,BASE_NO 3,IPO_FRAME #BASE,POINT2[] " "}
DECL E6POS Xl106={X 2229.7561,Y 132.126297,Z 331.531189,A 90.1379471,B -75.2002335,C 90.0486832,S 2,T 35,E1 -4300.01807,E2 0.0,E3 0.0,E4 0.0,E5 0.0,E6 0.0}
DECL FDAT Fl106={TOOL_NO 4,BASE_NO 3,IPO_FRAME #BASE,POINT2[] " "}
DECL PDAT Pvmax={VEL 100.0,ACC 100.0,APO_DIST 100.0}
DECL PDAT Pfin={VEL 100.0,ACC 100.0,APO_DIST 20.0,APO_MODE #CDIS}
DECL PDAT Pxlarge={VEL 100.0,ACC 100.0,APO_DIST 500.0,APO_MODE #CDIS}
DECL PDAT Pmedium={VEL 100.0,ACC 100.0,APO_DIST 100.0,APO_MODE #CDIS}
DECL PDAT Psmall={VEL 100.0,ACC 100.0,APO_DIST 50.0,APO_MODE #CDIS}
DECL PDAT Plarge={VEL 100.0,ACC 100.0,APO_DIST 200.0,APO_MODE #CDIS}
DECL E6POS Xl036={X 409.315002,Y 1105.31604,Z -10.6182203,A -174.052399,B 70.7239838,C 93.0403671,S 2,T 42,E1 -5500.00195,E2 0.0,E3 0.0,E4 0.0,E5 0.0,E6 0.0}
DECL FDAT Fl036={TOOL_NO 4,BASE_NO 3,IPO_FRAME #BASE,POINT2[] " "}
DECL E6POS Xl031={X 404.733307,Y 971.933472,Z -20.2303009,A -177.355896,B 65.1169662,C 90.2647705,S 2,T 43,E1 -5500.00195,E2 0.0,E3 0.0,E4 0.0,E5 0.0,E6 0.0}
DECL FDAT Fl031={TOOL_NO 4,BASE_NO 3,IPO_FRAME #BASE,POINT2[] " "}
DECL E6POS Xl026={X 404.733307,Y 971.933472,Z -20.2303009,A -177.355896,B 65.1169662,C 90.2647705,S 2,T 43,E1 -5500.00195,E2 0.0,E3 0.0,E4 0.0,E5 0.0,E6 0.0}
DECL FDAT Fl026={TOOL_NO 4,BASE_NO 3,IPO_FRAME #BASE,POINT2[] " "}
DECL E6POS Xl021={X 409.315002,Y 1105.31604,Z -10.6182203,A -174.052399,B 70.7239838,C 93.0403671,S 2,T 42,E1 -5500.00195,E2 0.0,E3 0.0,E4 0.0,E5 0.0,E6 0.0}
DECL FDAT Fl021={TOOL_NO 4,BASE_NO 3,IPO_FRAME #BASE,POINT2[] " "}
DECL E6POS Xl187={X 304.738007,Y 1263.75403,Z -0.123290703,A 176.651398,B 16.1943398,C 85.3128281,S 2,T 10,E1 -5500.00098,E2 0.0,E3 0.0,E4 0.0,E5 0.0,E6 0.0}
DECL FDAT Fl187={TOOL_NO 4,BASE_NO 3,IPO_FRAME #BASE,POINT2[] " "}
DECL E6POS Xl188={X 287.734711,Y 1322.29504,Z 74.3398666,A 178.265198,B 38.29142,C 90.978981,S 2,T 10,E1 -5500.00195,E2 0.0,E3 0.0,E4 0.0,E5 0.0,E6 0.0}
DECL FDAT Fl188={TOOL_NO 4,BASE_NO 3,IPO_FRAME #BASE,POINT2[] " "}
DECL PDAT Pmediun={VEL 100.0,ACC 100.0,APO_DIST 20.0,APO_MODE #CDIS}
DECL E6POS Xl157={X 538.371094,Y 1206.05603,Z 1316.33997,A -175.369995,B -40.4559517,C 83.8549881,S 2,T 10,E1 -5500.0,E2 0.0,E3 0.0,E4 0.0,E5 0.0,E6 0.0}
DECL FDAT Fl157={TOOL_NO 4,BASE_NO 3,IPO_FRAME #BASE,POINT2[] " "}
DECL E6POS Xl158={X 589.629211,Y 943.226929,Z 1281.97595,A -171.682404,B -45.6992912,C 81.6588135,S 2,T 11,E1 -5500.0,E2 0.0,E3 0.0,E4 0.0,E5 0.0,E6 0.0}
DECL FDAT Fl158={TOOL_NO 4,BASE_NO 3,IPO_FRAME #BASE,POINT2[] " "}
DECL E6POS Xl159={X 678.558472,Y 954.306213,Z 1295.41003,A -119.195297,B -83.508667,C 30.5657806,S 2,T 11,E1 -5500.0,E2 0.0,E3 0.0,E4 0.0,E5 0.0,E6 0.0}
DECL FDAT Fl159={TOOL_NO 4,BASE_NO 3,IPO_FRAME #BASE,POINT2[] " "}
DECL E6POS Xl161={X 671.624817,Y 1332.23401,Z 1295.65002,A -120.261002,B -83.4203491,C 31.5994892,S 2,T 10,E1 -5500.0,E2 0.0,E3 0.0,E4 0.0,E5 0.0,E6 0.0}
DECL FDAT Fl161={TOOL_NO 4,BASE_NO 3,IPO_FRAME #BASE,POINT2[] " "}
DECL E6POS Xl162={X 927.369385,Y 1296.62805,Z 1303.91895,A -120.261002,B -83.4203491,C 31.5994701,S 2,T 10,E1 -5500.0,E2 0.0,E3 0.0,E4 0.0,E5 0.0,E6 0.0}
DECL FDAT Fl162={TOOL_NO 4,BASE_NO 3,IPO_FRAME #BASE,POINT2[] " "}
DECL E6POS Xl163={X 954.363403,Y 959.226379,Z 1309.59399,A -12.1939201,B -68.716217,C -75.5949097,S 2,T 11,E1 -5500.0,E2 0.0,E3 0.0,E4 0.0,E5 0.0,E6 0.0}
DECL FDAT Fl163={TOOL_NO 4,BASE_NO 3,IPO_FRAME #BASE,POINT2[] " "}
DECL E6POS Xl164={X 954.363403,Y 959.226379,Z 1309.59399,A -12.1939201,B -68.716217,C -75.5949097,S 2,T 11,E1 -5500.0,E2 0.0,E3 0.0,E4 0.0,E5 0.0,E6 0.0}
DECL FDAT Fl164={TOOL_NO 4,BASE_NO 3,IPO_FRAME #BASE,POINT2[] " "}
DECL E6POS Xl166={X 954.106018,Y 1102.29199,Z 1310.23706,A -12.1939898,B -68.7160492,C -75.594841,S 2,T 10,E1 -5500.0,E2 0.0,E3 0.0,E4 0.0,E5 0.0,E6 0.0}
DECL FDAT Fl166={TOOL_NO 4,BASE_NO 3,IPO_FRAME #BASE,POINT2[] " "}
DECL E6POS Xl116={X 1120.76404,Y 1693.40405,Z 465.043793,A -103.135002,B -54.4802704,C 7.35247707,S 2,T 10,E1 -5500.0,E2 0.0,E3 0.0,E4 0.0,E5 0.0,E6 0.0}
DECL FDAT Fl116={TOOL_NO 4,BASE_NO 3,IPO_FRAME #BASE,POINT2[] " "}
DECL E6POS Xl171={X 493.426605,Y 954.01123,Z 1196.677,A -165.408203,B -64.9694595,C 76.488472,S 2,T 11,E1 -5500.0,E2 0.0,E3 0.0,E4 0.0,E5 0.0,E6 0.0}
DECL FDAT Fl171={TOOL_NO 4,BASE_NO 3,IPO_FRAME #BASE,POINT2[] " "}
DECL PDAT Pxxlarge={VEL 100.0,ACC 100.0,APO_DIST 1000.0,APO_MODE #CDIS}
DECL E6POS Xl527={X 3354.73999,Y 2478.89404,Z 10.7530003,A -163.420303,B -21.2028999,C -0.973699987,S 2,T 11,E1 -3400.0,E2 0.0,E3 0.0,E4 0.0,E5 0.0,E6 0.0}
DECL FDAT Fl527={TOOL_NO 4,BASE_NO 3,IPO_FRAME #BASE,POINT2[] " "}
ENDDAT
